LIN {X 0,Y 356.763,Z 514.388,A -85,B 0,C 180,E1 -13395.162,E2 -13395.162} C_VEL
LIN {X 0,Y 355.871,Z 522.553,A -85,B 0,C 180,E1 -13396.583,E2 -13396.583} C_VEL
LIN {X 0,Y 354.826,Z 530.602,A -85,B 0,C 180,E1 -13398.287,E2 -13398.287} C_VEL
LIN {X 0,Y 354.238,Z 536.073,A -85,B 0,C 180,E1 -13399.715,E2 -13399.715} C_VEL
LIN {X 0,Y 353.729,Z 541.453,A -85,B 0,C 180,E1 -13401.431,E2 -13401.431} C_VEL
LIN {X 0,Y 353.417,Z 545.66,A -85,B 0,C 180,E1 -13403.148,E2 -13403.148} C_VEL
LIN {X 0,Y 353.31,Z 547.883,A -85,B 0,C 180,E1 -13404.292,E2 -13404.292} C_VEL
LIN {X 0,Y 353.281,Z 549.633,A -85,B 0,C 180,E1 -13405.436,E2 -13405.436} C_VEL
LIN {X 0,Y 353.226,Z 550.976,A -85,B 0,C 180,E1 -13406.578,E2 -13406.578} C_VEL
LIN {X 0,Y 353.205,Z 551.922,A -85,B 0,C 180,E1 -13407.72,E2 -13407.72} C_VEL
LIN {X 0,Y 353.285,Z 552.443,A -85,B 0,C 180,E1 -13408.861,E2 -13408.861} C_VEL
LIN {X 0,Y 353.33,Z 552.542,A -85,B 0,C 180,E1 -13410,E2 -13410} C_VEL
LIN {X 0,Y 353.29,Z 552.246,A -85,B 0,C 180,E1 -13411.14,E2 -13411.14} C_VEL
LIN {X 0,Y 353.224,Z 551.556,A -85,B 0,C 180,E1 -13412.281,E2 -13412.281} C_VEL
LIN {X 0,Y 353.234,Z 550.435,A -85,B 0,C 180,E1 -13413.422,E2 -13413.422} C_VEL
LIN {X 0,Y 353.284,Z 548.872,A -85,B 0,C 180,E1 -13414.564,E2 -13414.564} C_VEL
LIN {X 0,Y 353.336,Z 545.71,A -85,B 0,C 180,E1 -13416.28,E2 -13416.28} C_VEL
LIN {X 0,Y 353.606,Z 541.468,A -85,B 0,C 180,E1 -13417.998,E2 -13417.998} C_VEL
LIN {X 0,Y 354.092,Z 535.01,A -85,B 0,C 180,E1 -13420.002,E2 -13420.002} C_VEL
LIN {X 0,Y 354.688,Z 527.935,A -85,B 0,C 180,E1 -13421.719,E2 -13421.719} C_VEL
LIN {X 0,Y 355.658,Z 519.093,A -85,B 0,C 180,E1 -13423.426,E2 -13423.426} C_VEL
LIN {X 0,Y 356.591,Z 510.04,A -85,B 0,C 180,E1 -13424.846,E2 -13424.846} C_VEL
LIN {X 0,Y 357.497,Z 500.082,A -85,B 0,C 180,E1 -13426.122,E2 -13426.122} C_VEL
LIN {X 0,Y 358.615,Z 489.083,A -85,B 0,C 180,E1 -13427.243,E2 -13427.243} C_VEL
LIN {X 0,Y 359.112,Z 482.478,A -85,B 0,C 180,E1 -13427.806,E2 -13427.806} C_VEL
LIN {X 0,Y 357.939,Z 470.567,A -85,B 0,C 180,E1 -13428.722,E2 -13428.722} C_VEL
LIN {X 0,Y 355.953,Z 457.17,A -85,B 0,C 180,E1 -13429.522,E2 -13429.522} C_VEL
LIN {X 0,Y 354.041,Z 446.07,A -85,B 0,C 180,E1 -13430.025,E2 -13430.025} C_VEL
LIN {X 0,Y 354.417,Z 439.879,A -85,B 0,C 180,E1 -13433.366,E2 -13433.366} C_VEL
LIN {X 0,Y 354.958,Z 433.091,A -85,B 0,C 180,E1 -13437.09,E2 -13437.09} C_VEL
LIN {X 0,Y 355.662,Z 426.292,A -85,B 0,C 180,E1 -13440.915,E2 -13440.915} C_VEL
LIN {X 0,Y 356.375,Z 419.492,A -85,B 0,C 180,E1 -13444.883,E2 -13444.883} C_VEL
LIN {X 0,Y 356.335,Z 416.053,A -85,B 0,C 180,E1 -13446.981,E2 -13446.981} C_VEL
LIN {X 0,Y 355.859,Z 411.923,A -85,B 0,C 180,E1 -13449.626,E2 -13449.626} C_VEL
LIN {X 0,Y 354.857,Z 406.322,A -85,B 0,C 180,E1 -13453.44,E2 -13453.44} C_VEL
LIN {X 0,Y 354.795,Z 406.29,A -85,B 0,C 180,E1 -13457.663,E2 -13457.663} C_VEL
LIN {X 0,Y 354.817,Z 406.286,A -85,B 0,C 180,E1 -13460.666,E2 -13460.666} C_VEL
LIN {X 0,Y 354.823,Z 406.284,A -85,B 0,C 180,E1 -13464.301,E2 -13464.301} C_VEL
LIN {X 0,Y 354.788,Z 406.29,A -85,B 0,C 180,E1 -13467.667,E2 -13467.667} C_VEL
LIN {X 0,Y 354.87,Z 406.28,A -85,B 0,C 180,E1 -13470.621,E2 -13470.621} C_VEL
LIN {X 0,Y 354.9,Z 406.274,A -85,B 0,C 180,E1 -13474.173,E2 -13474.173} C_VEL
LIN {X 0,Y 354.836,Z 406.283,A -85,B 0,C 180,E1 -13477.894,E2 -13477.894} C_VEL
LIN {X 0,Y 354.923,Z 406.272,A -85,B 0,C 180,E1 -13481.892,E2 -13481.892} C_VEL
LIN {X 0,Y 354.944,Z 406.269,A -85,B 0,C 180,E1 -13485.981,E2 -13485.981} C_VEL
LIN {X 0,Y 354.979,Z 406.265,A -85,B 0,C 180,E1 -13489.736,E2 -13489.736} C_VEL
LIN {X 0,Y 355.115,Z 406.248,A -85,B 0,C 180,E1 -13492.037,E2 -13492.037} C_VEL
LIN {X 0,Y 355.093,Z 406.251,A -85,B 0,C 180,E1 -13494.321,E2 -13494.321} C_VEL
LIN {X 0,Y 355.244,Z 406.232,A -85,B 0,C 180,E1 -13497.732,E2 -13497.732} C_VEL
LIN {X 0,Y 355.375,Z 406.215,A -85,B 0,C 180,E1 -13500,E2 -13500} C_VEL
LIN {X 0,Y 355.244,Z 406.232,A -85,B 0,C 180,E1 -13502.268,E2 -13502.268} C_VEL
LIN {X 0,Y 355.139,Z 406.25,A -85,B 0,C 180,E1 -13506.819,E2 -13506.819} C_VEL
LIN {X 0,Y 355.016,Z 406.264,A -85,B 0,C 180,E1 -13509.112,E2 -13509.112} C_VEL
LIN {X 0,Y 354.922,Z 406.275,A -85,B 0,C 180,E1 -13512.581,E2 -13512.581} C_VEL
LIN {X 0,Y 354.89,Z 406.276,A -85,B 0,C 180,E1 -13516.096,E2 -13516.096} C_VEL
LIN {X 0,Y 354.907,Z 406.277,A -85,B 0,C 180,E1 -13518.472,E2 -13518.472} C_VEL
LIN {X 0,Y 354.835,Z 406.283,A -85,B 0,C 180,E1 -13522.106,E2 -13522.106} C_VEL
LIN {X 0,Y 354.9,Z 406.274,A -85,B 0,C 180,E1 -13525.827,E2 -13525.827} C_VEL
LIN {X 0,Y 354.855,Z 406.28,A -85,B 0,C 180,E1 -13529.678,E2 -13529.678} C_VEL
LIN {X 0,Y 354.807,Z 406.286,A -85,B 0,C 180,E1 -13533.702,E2 -13533.702} C_VEL
LIN {X 0,Y 354.799,Z 406.291,A -85,B 0,C 180,E1 -13536.459,E2 -13536.459} C_VEL
LIN {X 0,Y 354.825,Z 406.284,A -85,B 0,C 180,E1 -13539.424,E2 -13539.424} C_VEL
LIN {X 0,Y 354.789,Z 406.292,A -85,B 0,C 180,E1 -13542.867,E2 -13542.867} C_VEL
LIN {X 0,Y 354.768,Z 406.293,A -85,B 0,C 180,E1 -13546.104,E2 -13546.104} C_VEL
LIN {X 0,Y 354.789,Z 406.289,A -85,B 0,C 180,E1 -13549.179,E2 -13549.179} C_VEL
LIN {X 0,Y 354.813,Z 406.29,A -85,B 0,C 180,E1 -13552.401,E2 -13552.401} C_VEL
LIN {X 0,Y 354.813,Z 406.287,A -85,B 0,C 180,E1 -13554.941,E2 -13554.941} C_VEL
LIN {X 0,Y 354.795,Z 406.292,A -85,B 0,C 180,E1 -13558.405,E2 -13558.405} C_VEL
LIN {X 0,Y 354.848,Z 406.281,A -85,B 0,C 180,E1 -13561.619,E2 -13561.619} C_VEL
LIN {X 0,Y 354.901,Z 406.278,A -85,B 0,C 180,E1 -13564.172,E2 -13564.172} C_VEL
LIN {X 0,Y 354.837,Z 406.283,A -85,B 0,C 180,E1 -13567.894,E2 -13567.894} C_VEL
LIN {X 0,Y 354.924,Z 406.273,A -85,B 0,C 180,E1 -13571.891,E2 -13571.891} C_VEL
LIN {X 0,Y 354.945,Z 406.271,A -85,B 0,C 180,E1 -13575.981,E2 -13575.981} C_VEL
LIN {X 0,Y 354.98,Z 406.265,A -85,B 0,C 180,E1 -13579.736,E2 -13579.736} C_VEL
LIN {X 0,Y 355.13,Z 406.249,A -85,B 0,C 180,E1 -13582.037,E2 -13582.037} C_VEL
LIN {X 0,Y 355.094,Z 406.255,A -85,B 0,C 180,E1 -13584.32,E2 -13584.32} C_VEL
LIN {X 0,Y 355.245,Z 406.233,A -85,B 0,C 180,E1 -13587.732,E2 -13587.732} C_VEL
LIN {X 0,Y 355.398,Z 406.216,A -85,B 0,C 180,E1 -13590,E2 -13590} C_VEL
LIN {X 0,Y 355.247,Z 406.237,A -85,B 0,C 180,E1 -13592.267,E2 -13592.267} C_VEL
LIN {X 0,Y 355.012,Z 406.261,A -85,B 0,C 180,E1 -13596.821,E2 -13596.821} C_VEL
LIN {X 0,Y 354.598,Z 406.315,A -85,B 0,C 180,E1 -13599.123,E2 -13599.123} C_VEL
LIN {X 0,Y 354.401,Z 408.438,A -85,B 0,C 180,E1 -13601.437,E2 -13601.437} C_VEL
LIN {X 0,Y 354.324,Z 410.917,A -85,B 0,C 180,E1 -13603.769,E2 -13603.769} C_VEL
LIN {X 0,Y 353.999,Z 415.198,A -85,B 0,C 180,E1 -13607.645,E2 -13607.645} C_VEL
LIN {X 0,Y 353.774,Z 418.936,A -85,B 0,C 180,E1 -13610.982,E2 -13610.982} C_VEL
LIN {X 0,Y 353.738,Z 421.29,A -85,B 0,C 180,E1 -13613.064,E2 -13613.064} C_VEL
LIN {X 0,Y 357.033,Z 435.378,A -85,B 0,C 180,E1 -13613.82,E2 -13613.82} C_VEL
LIN {X 0,Y 359.655,Z 448.278,A -85,B 0,C 180,E1 -13614.725,E2 -13614.725} C_VEL
LIN {X 0,Y 359.97,Z 452.375,A -85,B 0,C 180,E1 -13615.045,E2 -13615.045} C_VEL
LIN {X 0,Y 359.041,Z 463.653,A -85,B 0,C 180,E1 -13615.987,E2 -13615.987} C_VEL
LIN {X 0,Y 358.117,Z 474.495,A -85,B 0,C 180,E1 -13617.143,E2 -13617.143} C_VEL
LIN {X 0,Y 357.036,Z 484.857,A -85,B 0,C 180,E1 -13618.511,E2 -13618.511} C_VEL
LIN {X 0,Y 356.174,Z 493.935,A -85,B 0,C 180,E1 -13619.996,E2 -13619.996} C_VEL
LIN {X 0,Y 355.216,Z 502.345,A -85,B 0,C 180,E1 -13621.705,E2 -13621.705} C_VEL
LIN {X 0,Y 354.472,Z 509.826,A -85,B 0,C 180,E1 -13623.621,E2 -13623.621} C_VEL
LIN {X 0,Y 353.925,Z 515.495,A -85,B 0,C 180,E1 -13625.496,E2 -13625.496} C_VEL
LIN {X 0,Y 353.554,Z 519.696,A -85,B 0,C 180,E1 -13627.333,E2 -13627.333} C_VEL
LIN {X 0,Y 353.22,Z 523.205,A -85,B 0,C 180,E1 -13629.545,E2 -13629.545} C_VEL
LIN {X 0,Y 353.079,Z 524.676,A -85,B 0,C 180,E1 -13631.06,E2 -13631.06} C_VEL
LIN {X 0,Y 353.061,Z 525.477,A -85,B 0,C 180,E1 -13633.092,E2 -13633.092} C_VEL
LIN {X 0,Y 352.387,Z 525.561,A -85,B 0,C 180,E1 -13634.046,E2 -13634.046} C_VEL
LIN {X 0,Y 349.592,Z 525.045,A -85,B 0,C 180,E1 -13635.601,E2 -13635.601} C_VEL
LIN {X 0,Y 347.312,Z 524.205,A -85,B 0,C 180,E1 -13636.849,E2 -13636.849} C_VEL
LIN {X 0,Y 346.432,Z 523.164,A -85,B 0,C 180,E1 -13637.803,E2 -13637.803} C_VEL
LIN {X 0,Y 346.413,Z 522.725,A -85,B 0,C 180,E1 -13638.122,E2 -13638.122} C_VEL
LIN {X 0,Y 346.949,Z 518.902,A -85,B 0,C 180,E1 -13640.33,E2 -13640.33} C_VEL
LIN {X 0,Y 347.441,Z 514.693,A -85,B 0,C 180,E1 -13642.081,E2 -13642.081} C_VEL
LIN {X 0,Y 348.213,Z 509.279,A -85,B 0,C 180,E1 -13643.834,E2 -13643.834} C_VEL
LIN {X 0,Y 349.253,Z 501.981,A -85,B 0,C 180,E1 -13645.706,E2 -13645.706} C_VEL
LIN {X 0,Y 350.358,Z 493.618,A -85,B 0,C 180,E1 -13647.403,E2 -13647.403} C_VEL
LIN {X 0,Y 351.688,Z 483.939,A -85,B 0,C 180,E1 -13648.982,E2 -13648.982} C_VEL
LIN {X 0,Y 353.009,Z 473.091,A -85,B 0,C 180,E1 -13650.393,E2 -13650.393} C_VEL
LIN {X 0,Y 354.223,Z 461.722,A -85,B 0,C 180,E1 -13651.564,E2 -13651.564} C_VEL
LIN {X 0,Y 354.923,Z 454.745,A -85,B 0,C 180,E1 -13652.156,E2 -13652.156} C_VEL
LIN {X 0,Y 353.362,Z 445.433,A -85,B 0,C 180,E1 -13652.972,E2 -13652.972} C_VEL
LIN {X 0,Y 350.233,Z 433.278,A -85,B 0,C 180,E1 -13653.923,E2 -13653.923} C_VEL
LIN {X 0,Y 347.022,Z 422.964,A -85,B 0,C 180,E1 -13654.63,E2 -13654.63} C_VEL
LIN {X 0,Y 347.299,Z 418.94,A -85,B 0,C 180,E1 -13658.639,E2 -13658.639} C_VEL
LIN {X 0,Y 347.622,Z 415.352,A -85,B 0,C 180,E1 -13662.346,E2 -13662.346} C_VEL
LIN {X 0,Y 347.97,Z 411.993,A -85,B 0,C 180,E1 -13665.974,E2 -13665.974} C_VEL
LIN {X 0,Y 348.063,Z 408.92,A -85,B 0,C 180,E1 -13669.53,E2 -13669.53} C_VEL
LIN {X 0,Y 348.075,Z 407.133,A -85,B 0,C 180,E1 -13671.875,E2 -13671.875} C_VEL
LIN {X 0,Y 348.064,Z 407.131,A -85,B 0,C 180,E1 -13674.206,E2 -13674.206} C_VEL
LIN {X 0,Y 348.205,Z 407.115,A -85,B 0,C 180,E1 -13677.687,E2 -13677.687} C_VEL
LIN {X 0,Y 348.365,Z 407.093,A -85,B 0,C 180,E1 -13680,E2 -13680} C_VEL
LIN {X 0,Y 348.204,Z 407.11,A -85,B 0,C 180,E1 -13682.314,E2 -13682.314} C_VEL
LIN {X 0,Y 348.102,Z 407.126,A -85,B 0,C 180,E1 -13686.958,E2 -13686.958} C_VEL
LIN {X 0,Y 347.963,Z 407.142,A -85,B 0,C 180,E1 -13689.299,E2 -13689.299} C_VEL
LIN {X 0,Y 347.886,Z 407.153,A -85,B 0,C 180,E1 -13692.84,E2 -13692.84} C_VEL
LIN {X 0,Y 347.835,Z 407.16,A -85,B 0,C 180,E1 -13696.432,E2 -13696.432} C_VEL
LIN {X 0,Y 347.852,Z 407.156,A -85,B 0,C 180,E1 -13698.861,E2 -13698.861} C_VEL
LIN {X 0,Y 347.771,Z 407.167,A -85,B 0,C 180,E1 -13702.58,E2 -13702.58} C_VEL
LIN {X 0,Y 347.809,Z 407.162,A -85,B 0,C 180,E1 -13705.109,E2 -13705.109} C_VEL
LIN {X 0,Y 347.809,Z 407.163,A -85,B 0,C 180,E1 -13707.694,E2 -13707.694} C_VEL
LIN {X 0,Y 347.761,Z 407.168,A -85,B 0,C 180,E1 -13710.347,E2 -13710.347} C_VEL
LIN {X 0,Y 347.742,Z 407.171,A -85,B 0,C 180,E1 -13714.464,E2 -13714.464} C_VEL
LIN {X 0,Y 347.777,Z 407.169,A -85,B 0,C 180,E1 -13717.99,E2 -13717.99} C_VEL
LIN {X 0,Y 347.764,Z 407.171,A -85,B 0,C 180,E1 -13721.828,E2 -13721.828} C_VEL
LIN {X 0,Y 347.778,Z 407.283,A -85,B 0,C 180,E1 -13722.963,E2 -13722.963} C_VEL
LIN {X 0,Y 348.497,Z 411.314,A -85,B 0,C 180,E1 -13726.713,E2 -13726.713} C_VEL
LIN {X 0,Y 349.142,Z 415.165,A -85,B 0,C 180,E1 -13729.9,E2 -13729.9} C_VEL
LIN {X 0,Y 349.675,Z 419.167,A -85,B 0,C 180,E1 -13732.919,E2 -13732.919} C_VEL
LIN {X 0,Y 349.503,Z 423.291,A -85,B 0,C 180,E1 -13735.735,E2 -13735.735} C_VEL
LIN {X 0,Y 348.599,Z 429.618,A -85,B 0,C 180,E1 -13739.735,E2 -13739.735} C_VEL
LIN {X 0,Y 347.89,Z 436.102,A -85,B 0,C 180,E1 -13743.613,E2 -13743.613} C_VEL
LIN {X 0,Y 347.341,Z 442.681,A -85,B 0,C 180,E1 -13747.392,E2 -13747.392} C_VEL
LIN {X 0,Y 347.201,Z 444.613,A -85,B 0,C 180,E1 -13748.408,E2 -13748.408} C_VEL
LIN {X 0,Y 350.304,Z 458.15,A -85,B 0,C 180,E1 -13749.191,E2 -13749.191} C_VEL
LIN {X 0,Y 352.434,Z 470.851,A -85,B 0,C 180,E1 -13750.101,E2 -13750.101} C_VEL
LIN {X 0,Y 353.332,Z 482.24,A -85,B 0,C 180,E1 -13751.055,E2 -13751.055} C_VEL
LIN {X 0,Y 353.175,Z 487.99,A -85,B 0,C 180,E1 -13751.585,E2 -13751.585} C_VEL
LIN {X 0,Y 351.873,Z 498.895,A -85,B 0,C 180,E1 -13752.717,E2 -13752.717} C_VEL
LIN {X 0,Y 350.628,Z 508.537,A -85,B 0,C 180,E1 -13753.962,E2 -13753.962} C_VEL
LIN {X 0,Y 349.561,Z 517.851,A -85,B 0,C 180,E1 -13755.445,E2 -13755.445} C_VEL
LIN {X 0,Y 348.374,Z 526.733,A -85,B 0,C 180,E1 -13757.179,E2 -13757.179} C_VEL
LIN {X 0,Y 347.438,Z 533.896,A -85,B 0,C 180,E1 -13758.921,E2 -13758.921} C_VEL
LIN {X 0,Y 346.854,Z 539.65,A -85,B 0,C 180,E1 -13760.672,E2 -13760.672} C_VEL
LIN {X 0,Y 346.464,Z 544.204,A -85,B 0,C 180,E1 -13762.424,E2 -13762.424} C_VEL
LIN {X 0,Y 346.23,Z 547.676,A -85,B 0,C 180,E1 -13764.175,E2 -13764.175} C_VEL
LIN {X 0,Y 346.179,Z 549.414,A -85,B 0,C 180,E1 -13765.343,E2 -13765.343} C_VEL
LIN {X 0,Y 346.15,Z 550.746,A -85,B 0,C 180,E1 -13766.508,E2 -13766.508} C_VEL
LIN {X 0,Y 346.114,Z 551.679,A -85,B 0,C 180,E1 -13767.673,E2 -13767.673} C_VEL
LIN {X 0,Y 346.186,Z 552.174,A -85,B 0,C 180,E1 -13768.837,E2 -13768.837} C_VEL
LIN {X 0,Y 346.235,Z 552.261,A -85,B 0,C 180,E1 -13770,E2 -13770} C_VEL
LIN {X 0,Y 346.192,Z 551.951,A -85,B 0,C 180,E1 -13771.164,E2 -13771.164} C_VEL
LIN {X 0,Y 346.132,Z 551.247,A -85,B 0,C 180,E1 -13772.328,E2 -13772.328} C_VEL
LIN {X 0,Y 346.157,Z 550.098,A -85,B 0,C 180,E1 -13773.492,E2 -13773.492} C_VEL
LIN {X 0,Y 346.174,Z 547.182,A -85,B 0,C 180,E1 -13775.463,E2 -13775.463} C_VEL
LIN {X 0,Y 346.444,Z 542.612,A -85,B 0,C 180,E1 -13777.577,E2 -13777.577} C_VEL
LIN {X 0,Y 346.788,Z 537.556,A -85,B 0,C 180,E1 -13779.331,E2 -13779.331} C_VEL
LIN {X 0,Y 347.323,Z 531.186,A -85,B 0,C 180,E1 -13781.083,E2 -13781.083} C_VEL
LIN {X 0,Y 348.226,Z 523.209,A -85,B 0,C 180,E1 -13782.827,E2 -13782.827} C_VEL
LIN {X 0,Y 349.088,Z 515.082,A -85,B 0,C 180,E1 -13784.278,E2 -13784.278} C_VEL
LIN {X 0,Y 350.014,Z 505.606,A -85,B 0,C 180,E1 -13785.668,E2 -13785.668} C_VEL
LIN {X 0,Y 351.055,Z 495.486,A -85,B 0,C 180,E1 -13786.875,E2 -13786.875} C_VEL
LIN {X 0,Y 352.084,Z 485.062,A -85,B 0,C 180,E1 -13787.873,E2 -13787.873} C_VEL
LIN {X 0,Y 351.589,Z 476.667,A -85,B 0,C 180,E1 -13788.577,E2 -13788.577} C_VEL
LIN {X 0,Y 350.033,Z 464.231,A -85,B 0,C 180,E1 -13789.458,E2 -13789.458} C_VEL
LIN {X 0,Y 347.82,Z 450.648,A -85,B 0,C 180,E1 -13790.182,E2 -13790.182} C_VEL
LIN {X 0,Y 347.013,Z 445.844,A -85,B 0,C 180,E1 -13790.391,E2 -13790.391} C_VEL
LIN {X 0,Y 347.494,Z 438.444,A -85,B 0,C 180,E1 -13794.478,E2 -13794.478} C_VEL
LIN {X 0,Y 348.096,Z 431.644,A -85,B 0,C 180,E1 -13798.325,E2 -13798.325} C_VEL
LIN {X 0,Y 348.685,Z 425.984,A -85,B 0,C 180,E1 -13801.604,E2 -13801.604} C_VEL
LIN {X 0,Y 349.34,Z 420.319,A -85,B 0,C 180,E1 -13804.986,E2 -13804.986} C_VEL
LIN {X 0,Y 349.31,Z 416.89,A -85,B 0,C 180,E1 -13807.128,E2 -13807.128} C_VEL
LIN {X 0,Y 348.738,Z 412.487,A -85,B 0,C 180,E1 -13810.021,E2 -13810.021} C_VEL
LIN {X 0,Y 347.84,Z 407.486,A -85,B 0,C 180,E1 -13813.5,E2 -13813.5} C_VEL
LIN {X 0,Y 347.759,Z 407.169,A -85,B 0,C 180,E1 -13813.771,E2 -13813.771} C_VEL
LIN {X 0,Y 347.727,Z 407.171,A -85,B 0,C 180,E1 -13816.686,E2 -13816.686} C_VEL
LIN {X 0,Y 347.748,Z 407.165,A -85,B 0,C 180,E1 -13820.173,E2 -13820.173} C_VEL
LIN {X 0,Y 347.763,Z 407.165,A -85,B 0,C 180,E1 -13822.679,E2 -13822.679} C_VEL
LIN {X 0,Y 347.75,Z 407.165,A -85,B 0,C 180,E1 -13825.956,E2 -13825.956} C_VEL
LIN {X 0,Y 347.765,Z 407.165,A -85,B 0,C 180,E1 -13829.653,E2 -13829.653} C_VEL
LIN {X 0,Y 347.852,Z 407.155,A -85,B 0,C 180,E1 -13832.745,E2 -13832.745} C_VEL
LIN {X 0,Y 347.79,Z 407.16,A -85,B 0,C 180,E1 -13836.162,E2 -13836.162} C_VEL
LIN {X 0,Y 347.814,Z 407.157,A -85,B 0,C 180,E1 -13839.909,E2 -13839.909} C_VEL
LIN {X 0,Y 347.867,Z 407.151,A -85,B 0,C 180,E1 -13842.359,E2 -13842.359} C_VEL
LIN {X 0,Y 347.898,Z 407.146,A -85,B 0,C 180,E1 -13845.971,E2 -13845.971} C_VEL
LIN {X 0,Y 347.929,Z 407.144,A -85,B 0,C 180,E1 -13849.526,E2 -13849.526} C_VEL
LIN {X 0,Y 348.075,Z 407.125,A -85,B 0,C 180,E1 -13851.875,E2 -13851.875} C_VEL
LIN {X 0,Y 348.068,Z 407.126,A -85,B 0,C 180,E1 -13854.206,E2 -13854.206} C_VEL
LIN {X 0,Y 348.206,Z 407.109,A -85,B 0,C 180,E1 -13857.686,E2 -13857.686} C_VEL
LIN {X 0,Y 348.326,Z 407.093,A -85,B 0,C 180,E1 -13860,E2 -13860} C_VEL
LIN {X 0,Y 348.206,Z 407.109,A -85,B 0,C 180,E1 -13862.313,E2 -13862.313} C_VEL
LIN {X 0,Y 348.107,Z 407.126,A -85,B 0,C 180,E1 -13866.958,E2 -13866.958} C_VEL
LIN {X 0,Y 347.968,Z 407.14,A -85,B 0,C 180,E1 -13869.298,E2 -13869.298} C_VEL
LIN {X 0,Y 347.89,Z 407.153,A -85,B 0,C 180,E1 -13872.839,E2 -13872.839} C_VEL
LIN {X 0,Y 347.84,Z 407.156,A -85,B 0,C 180,E1 -13876.431,E2 -13876.431} C_VEL
LIN {X 0,Y 347.857,Z 407.157,A -85,B 0,C 180,E1 -13878.86,E2 -13878.86} C_VEL
LIN {X 0,Y 347.775,Z 407.166,A -85,B 0,C 180,E1 -13882.579,E2 -13882.579} C_VEL
LIN {X 0,Y 347.813,Z 407.16,A -85,B 0,C 180,E1 -13885.108,E2 -13885.108} C_VEL
LIN {X 0,Y 347.812,Z 407.157,A -85,B 0,C 180,E1 -13887.694,E2 -13887.694} C_VEL
LIN {X 0,Y 347.765,Z 407.166,A -85,B 0,C 180,E1 -13890.346,E2 -13890.346} C_VEL
LIN {X 0,Y 347.745,Z 407.169,A -85,B 0,C 180,E1 -13894.464,E2 -13894.464} C_VEL
LIN {X 0,Y 347.774,Z 407.162,A -85,B 0,C 180,E1 -13897.989,E2 -13897.989} C_VEL
LIN {X 0,Y 347.751,Z 407.165,A -85,B 0,C 180,E1 -13901.83,E2 -13901.83} C_VEL
LIN {X 0,Y 347.706,Z 407.173,A -85,B 0,C 180,E1 -13905.027,E2 -13905.027} C_VEL
LIN {X 0,Y 347.751,Z 407.169,A -85,B 0,C 180,E1 -13908.397,E2 -13908.397} C_VEL
LIN {X 0,Y 347.778,Z 407.163,A -85,B 0,C 180,E1 -13912.011,E2 -13912.011} C_VEL
LIN {X 0,Y 347.746,Z 407.165,A -85,B 0,C 180,E1 -13915.536,E2 -13915.536} C_VEL
LIN {X 0,Y 347.746,Z 407.169,A -85,B 0,C 180,E1 -13918.3,E2 -13918.3} C_VEL
LIN {X 0,Y 347.78,Z 407.163,A -85,B 0,C 180,E1 -13920.988,E2 -13920.988} C_VEL
LIN {X 0,Y 347.832,Z 407.155,A -85,B 0,C 180,E1 -13923.608,E2 -13923.608} C_VEL
LIN {X 0,Y 347.791,Z 407.163,A -85,B 0,C 180,E1 -13926.162,E2 -13926.162} C_VEL
LIN {X 0,Y 347.815,Z 407.158,A -85,B 0,C 180,E1 -13929.909,E2 -13929.909} C_VEL
LIN {X 0,Y 347.868,Z 407.156,A -85,B 0,C 180,E1 -13932.359,E2 -13932.359} C_VEL
LIN {X 0,Y 347.899,Z 407.149,A -85,B 0,C 180,E1 -13935.971,E2 -13935.971} C_VEL
LIN {X 0,Y 347.93,Z 407.142,A -85,B 0,C 180,E1 -13939.525,E2 -13939.525} C_VEL
LIN {X 0,Y 348.11,Z 407.121,A -85,B 0,C 180,E1 -13943.042,E2 -13943.042} C_VEL
LIN {X 0,Y 348.207,Z 407.109,A -85,B 0,C 180,E1 -13947.686,E2 -13947.686} C_VEL
LIN {X 0,Y 348.346,Z 407.094,A -85,B 0,C 180,E1 -13950,E2 -13950} C_VEL
LIN {X 0,Y 348.209,Z 407.113,A -85,B 0,C 180,E1 -13952.313,E2 -13952.313} C_VEL
LIN {X 0,Y 348.02,Z 407.133,A -85,B 0,C 180,E1 -13955.795,E2 -13955.795} C_VEL
LIN {X 0,Y 347.736,Z 407.172,A -85,B 0,C 180,E1 -13958.133,E2 -13958.133} C_VEL
LIN {X 0,Y 347.524,Z 407.196,A -85,B 0,C 180,E1 -13959.31,E2 -13959.31} C_VEL
LIN {X 0,Y 347.326,Z 410.762,A -85,B 0,C 180,E1 -13962.86,E2 -13962.86} C_VEL
LIN {X 0,Y 346.985,Z 414.642,A -85,B 0,C 180,E1 -13966.472,E2 -13966.472} C_VEL
LIN {X 0,Y 346.739,Z 418.725,A -85,B 0,C 180,E1 -13970.155,E2 -13970.155} C_VEL
LIN {X 0,Y 346.638,Z 421.563,A -85,B 0,C 180,E1 -13972.696,E2 -13972.696} C_VEL
LIN {X 0,Y 350.042,Z 435.676,A -85,B 0,C 180,E1 -13973.478,E2 -13973.478} C_VEL
LIN {X 0,Y 352.692,Z 448.785,A -85,B 0,C 180,E1 -13974.423,E2 -13974.423} C_VEL
LIN {X 0,Y 353.121,Z 453.224,A -85,B 0,C 180,E1 -13974.783,E2 -13974.783} C_VEL
LIN {X 0,Y 352.177,Z 464.157,A -85,B 0,C 180,E1 -13975.724,E2 -13975.724} C_VEL
LIN {X 0,Y 351.175,Z 475.125,A -85,B 0,C 180,E1 -13976.922,E2 -13976.922} C_VEL
LIN {X 0,Y 350.016,Z 485.905,A -85,B 0,C 180,E1 -13978.388,E2 -13978.388} C_VEL
LIN {X 0,Y 349.057,Z 495.466,A -85,B 0,C 180,E1 -13980.029,E2 -13980.029} C_VEL
LIN {X 0,Y 348.144,Z 503.166,A -85,B 0,C 180,E1 -13981.658,E2 -13981.658} C_VEL
LIN {X 0,Y 347.429,Z 510.191,A -85,B 0,C 180,E1 -13983.51,E2 -13983.51} C_VEL
LIN {X 0,Y 346.911,Z 515.218,A -85,B 0,C 180,E1 -13985.184,E2 -13985.184} C_VEL
LIN {X 0,Y 346.556,Z 518.912,A -85,B 0,C 180,E1 -13986.744,E2 -13986.744} C_VEL
LIN {X 0,Y 346.328,Z 521.77,A -85,B 0,C 180,E1 -13988.302,E2 -13988.302} C_VEL
LIN {X 0,Y 346.025,Z 524.54,A -85,B 0,C 180,E1 -13990.536,E2 -13990.536} C_VEL
LIN {X 0,Y 345.996,Z 525.535,A -85,B 0,C 180,E1 -13992.09,E2 -13992.09} C_VEL
LIN {X 0,Y 345.984,Z 525.845,A -85,B 0,C 180,E1 -13993.68,E2 -13993.68} C_VEL
LIN {X 0,Y 346.028,Z 525.406,A -85,B 0,C 180,E1 -13995.304,E2 -13995.304} C_VEL
LIN {X 0,Y 346.213,Z 524.128,A -85,B 0,C 180,E1 -13996.951,E2 -13996.951} C_VEL
LIN {X 0,Y 346.413,Z 522.725,A -85,B 0,C 180,E1 -13998.122,E2 -13998.122} C_VEL
LIN {X 0,Y 345.957,Z 521.356,A -85,B 0,C 180,E1 -13999.069,E2 -13999.069} C_VEL
LIN {X 0,Y 343.495,Z 518.707,A -85,B 0,C 180,E1 -14000.606,E2 -14000.606} C_VEL
LIN {X 0,Y 341.465,Z 516.174,A -85,B 0,C 180,E1 -14001.823,E2 -14001.823} C_VEL
LIN {X 0,Y 340.763,Z 513.872,A -85,B 0,C 180,E1 -14002.732,E2 -14002.732} C_VEL
LIN {X 0,Y 340.8,Z 512.997,A -85,B 0,C 180,E1 -14003.03,E2 -14003.03} C_VEL
LIN {X 0,Y 341.628,Z 507.032,A -85,B 0,C 180,E1 -14004.829,E2 -14004.829} C_VEL
LIN {X 0,Y 342.559,Z 500.753,A -85,B 0,C 180,E1 -14006.362,E2 -14006.362} C_VEL
LIN {X 0,Y 343.648,Z 493.227,A -85,B 0,C 180,E1 -14007.878,E2 -14007.878} C_VEL
LIN {X 0,Y 345.004,Z 484.056,A -85,B 0,C 180,E1 -14009.385,E2 -14009.385} C_VEL
LIN {X 0,Y 346.32,Z 473.681,A -85,B 0,C 180,E1 -14010.762,E2 -14010.762} C_VEL
LIN {X 0,Y 347.596,Z 462.356,A -85,B 0,C 180,E1 -14011.96,E2 -14011.96} C_VEL
LIN {X 0,Y 348.27,Z 456.14,A -85,B 0,C 180,E1 -14012.504,E2 -14012.504} C_VEL
LIN {X 0,Y 346.435,Z 445.399,A -85,B 0,C 180,E1 -14013.493,E2 -14013.493} C_VEL
LIN {X 0,Y 343.142,Z 433.06,A -85,B 0,C 180,E1 -14014.485,E2 -14014.485} C_VEL
LIN {X 0,Y 339.984,Z 423.278,A -85,B 0,C 180,E1 -14015.195,E2 -14015.195} C_VEL
LIN {X 0,Y 340.315,Z 419.114,A -85,B 0,C 180,E1 -14019.447,E2 -14019.447} C_VEL
LIN {X 0,Y 340.665,Z 415.59,A -85,B 0,C 180,E1 -14023.213,E2 -14023.213} C_VEL
LIN {X 0,Y 340.982,Z 412.316,A -85,B 0,C 180,E1 -14026.896,E2 -14026.896} C_VEL
LIN {X 0,Y 341.072,Z 409.317,A -85,B 0,C 180,E1 -14030.512,E2 -14030.512} C_VEL
LIN {X 0,Y 341.083,Z 408.364,A -85,B 0,C 180,E1 -14031.707,E2 -14031.707} C_VEL
LIN {X 0,Y 341.073,Z 408.002,A -85,B 0,C 180,E1 -14032.898,E2 -14032.898} C_VEL
LIN {X 0,Y 341.166,Z 407.991,A -85,B 0,C 180,E1 -14037.639,E2 -14037.639} C_VEL
LIN {X 0,Y 341.314,Z 407.972,A -85,B 0,C 180,E1 -14040,E2 -14040} C_VEL
LIN {X 0,Y 341.166,Z 407.987,A -85,B 0,C 180,E1 -14042.361,E2 -14042.361} C_VEL
LIN {X 0,Y 341.072,Z 408.001,A -85,B 0,C 180,E1 -14047.102,E2 -14047.102} C_VEL
LIN {X 0,Y 340.867,Z 408.026,A -85,B 0,C 180,E1 -14050.694,E2 -14050.694} C_VEL
LIN {X 0,Y 340.859,Z 408.028,A -85,B 0,C 180,E1 -14054.325,E2 -14054.325} C_VEL
LIN {X 0,Y 340.834,Z 408.03,A -85,B 0,C 180,E1 -14058.467,E2 -14058.467} C_VEL
LIN {X 0,Y 340.75,Z 408.041,A -85,B 0,C 180,E1 -14061.857,E2 -14061.857} C_VEL
LIN {X 0,Y 340.77,Z 408.039,A -85,B 0,C 180,E1 -14065.665,E2 -14065.665} C_VEL
LIN {X 0,Y 340.739,Z 408.042,A -85,B 0,C 180,E1 -14068.32,E2 -14068.32} C_VEL
LIN {X 0,Y 340.701,Z 408.048,A -85,B 0,C 180,E1 -14071.045,E2 -14071.045} C_VEL
LIN {X 0,Y 340.716,Z 408.048,A -85,B 0,C 180,E1 -14075.279,E2 -14075.279} C_VEL
LIN {X 0,Y 340.717,Z 408.049,A -85,B 0,C 180,E1 -14078.389,E2 -14078.389} C_VEL
LIN {X 0,Y 340.715,Z 408.051,A -85,B 0,C 180,E1 -14082.189,E2 -14082.189} C_VEL
LIN {X 0,Y 341.42,Z 412.084,A -85,B 0,C 180,E1 -14086.093,E2 -14086.093} C_VEL
LIN {X 0,Y 342.063,Z 416.006,A -85,B 0,C 180,E1 -14089.482,E2 -14089.482} C_VEL
LIN {X 0,Y 342.554,Z 419.218,A -85,B 0,C 180,E1 -14092.013,E2 -14092.013} C_VEL
LIN {X 0,Y 342.665,Z 422.257,A -85,B 0,C 180,E1 -14094.231,E2 -14094.231} C_VEL
LIN {X 0,Y 342.018,Z 427.441,A -85,B 0,C 180,E1 -14097.707,E2 -14097.707} C_VEL
LIN {X 0,Y 341.166,Z 433.826,A -85,B 0,C 180,E1 -14101.72,E2 -14101.72} C_VEL
LIN {X 0,Y 340.517,Z 440.346,A -85,B 0,C 180,E1 -14105.621,E2 -14105.621} C_VEL
LIN {X 0,Y 340.245,Z 444.312,A -85,B 0,C 180,E1 -14107.857,E2 -14107.857} C_VEL
LIN {X 0,Y 343.432,Z 457.952,A -85,B 0,C 180,E1 -14108.677,E2 -14108.677} C_VEL
LIN {X 0,Y 345.501,Z 470.026,A -85,B 0,C 180,E1 -14109.572,E2 -14109.572} C_VEL
LIN {X 0,Y 346.495,Z 481.283,A -85,B 0,C 180,E1 -14110.543,E2 -14110.543} C_VEL
LIN {X 0,Y 346.453,Z 488.312,A -85,B 0,C 180,E1 -14111.215,E2 -14111.215} C_VEL
LIN {X 0,Y 345.101,Z 499.072,A -85,B 0,C 180,E1 -14112.367,E2 -14112.367} C_VEL
LIN {X 0,Y 343.778,Z 508.808,A -85,B 0,C 180,E1 -14113.661,E2 -14113.661} C_VEL
LIN {X 0,Y 342.669,Z 517.882,A -85,B 0,C 180,E1 -14115.146,E2 -14115.146} C_VEL
LIN {X 0,Y 341.439,Z 526.715,A -85,B 0,C 180,E1 -14116.914,E2 -14116.914} C_VEL
LIN {X 0,Y 340.43,Z 533.811,A -85,B 0,C 180,E1 -14118.69,E2 -14118.69} C_VEL
LIN {X 0,Y 339.808,Z 539.516,A -85,B 0,C 180,E1 -14120.477,E2 -14120.477} C_VEL
LIN {X 0,Y 339.395,Z 544.03,A -85,B 0,C 180,E1 -14122.265,E2 -14122.265} C_VEL
LIN {X 0,Y 339.135,Z 547.558,A -85,B 0,C 180,E1 -14124.11,E2 -14124.11} C_VEL
LIN {X 0,Y 339.074,Z 550.517,A -85,B 0,C 180,E1 -14126.435,E2 -14126.435} C_VEL
LIN {X 0,Y 339.027,Z 551.432,A -85,B 0,C 180,E1 -14127.624,E2 -14127.624} C_VEL
LIN {X 0,Y 339.087,Z 551.905,A -85,B 0,C 180,E1 -14128.813,E2 -14128.813} C_VEL
LIN {X 0,Y 339.14,Z 551.979,A -85,B 0,C 180,E1 -14130,E2 -14130} C_VEL
LIN {X 0,Y 339.094,Z 551.657,A -85,B 0,C 180,E1 -14131.188,E2 -14131.188} C_VEL
LIN {X 0,Y 339.043,Z 550.935,A -85,B 0,C 180,E1 -14132.376,E2 -14132.376} C_VEL
LIN {X 0,Y 339.082,Z 549.762,A -85,B 0,C 180,E1 -14133.565,E2 -14133.565} C_VEL
LIN {X 0,Y 339.094,Z 548.167,A -85,B 0,C 180,E1 -14134.756,E2 -14134.756} C_VEL
LIN {X 0,Y 339.194,Z 544.942,A -85,B 0,C 180,E1 -14136.544,E2 -14136.544} C_VEL
LIN {X 0,Y 339.477,Z 540.631,A -85,B 0,C 180,E1 -14138.333,E2 -14138.333} C_VEL
LIN {X 0,Y 340.043,Z 534.092,A -85,B 0,C 180,E1 -14140.419,E2 -14140.419} C_VEL
LIN {X 0,Y 340.749,Z 526.893,A -85,B 0,C 180,E1 -14142.205,E2 -14142.205} C_VEL
LIN {X 0,Y 341.738,Z 517.943,A -85,B 0,C 180,E1 -14143.984,E2 -14143.984} C_VEL
LIN {X 0,Y 342.687,Z 508.763,A -85,B 0,C 180,E1 -14145.463,E2 -14145.463} C_VEL
LIN {X 0,Y 343.785,Z 498.595,A -85,B 0,C 180,E1 -14146.784,E2 -14146.784} C_VEL
LIN {X 0,Y 345,Z 487.387,A -85,B 0,C 180,E1 -14147.946,E2 -14147.946} C_VEL
LIN {X 0,Y 345.118,Z 482.363,A -85,B 0,C 180,E1 -14148.4,E2 -14148.4} C_VEL
LIN {X 0,Y 343.888,Z 470.053,A -85,B 0,C 180,E1 -14149.397,E2 -14149.397} C_VEL
LIN {X 0,Y 341.902,Z 456.815,A -85,B 0,C 180,E1 -14150.233,E2 -14150.233} C_VEL
LIN {X 0,Y 339.957,Z 445.557,A -85,B 0,C 180,E1 -14150.783,E2 -14150.783} C_VEL
LIN {X 0,Y 340.457,Z 438.598,A -85,B 0,C 180,E1 -14154.73,E2 -14154.73} C_VEL
LIN {X 0,Y 341.157,Z 431.305,A -85,B 0,C 180,E1 -14158.955,E2 -14158.955} C_VEL
LIN {X 0,Y 341.771,Z 425.657,A -85,B 0,C 180,E1 -14162.32,E2 -14162.32} C_VEL
LIN {X 0,Y 342.33,Z 421.121,A -85,B 0,C 180,E1 -14165.088,E2 -14165.088} C_VEL
LIN {X 0,Y 342.165,Z 416.546,A -85,B 0,C 180,E1 -14168.039,E2 -14168.039} C_VEL
LIN {X 0,Y 341.427,Z 411.918,A -85,B 0,C 180,E1 -14171.201,E2 -14171.201} C_VEL
LIN {X 0,Y 340.711,Z 408.047,A -85,B 0,C 180,E1 -14173.999,E2 -14173.999} C_VEL
LIN {X 0,Y 340.7,Z 408.043,A -85,B 0,C 180,E1 -14177.955,E2 -14177.955} C_VEL
LIN {X 0,Y 340.734,Z 408.04,A -85,B 0,C 180,E1 -14181.773,E2 -14181.773} C_VEL
LIN {X 0,Y 340.724,Z 408.042,A -85,B 0,C 180,E1 -14185.595,E2 -14185.595} C_VEL
LIN {X 0,Y 340.705,Z 408.046,A -85,B 0,C 180,E1 -14188.956,E2 -14188.956} C_VEL
LIN {X 0,Y 340.779,Z 408.034,A -85,B 0,C 180,E1 -14192.474,E2 -14192.474} C_VEL
LIN {X 0,Y 340.757,Z 408.037,A -85,B 0,C 180,E1 -14195.638,E2 -14195.638} C_VEL
LIN {X 0,Y 340.746,Z 408.04,A -85,B 0,C 180,E1 -14199.474,E2 -14199.474} C_VEL
LIN {X 0,Y 340.859,Z 408.023,A -85,B 0,C 180,E1 -14201.984,E2 -14201.984} C_VEL
LIN {X 0,Y 340.87,Z 408.022,A -85,B 0,C 180,E1 -14205.705,E2 -14205.705} C_VEL
LIN {X 0,Y 340.872,Z 408.025,A -85,B 0,C 180,E1 -14209.306,E2 -14209.306} C_VEL
LIN {X 0,Y 341.076,Z 408.001,A -85,B 0,C 180,E1 -14212.898,E2 -14212.898} C_VEL
LIN {X 0,Y 341.168,Z 407.985,A -85,B 0,C 180,E1 -14217.639,E2 -14217.639} C_VEL
LIN {X 0,Y 341.277,Z 407.971,A -85,B 0,C 180,E1 -14220,E2 -14220} C_VEL
LIN {X 0,Y 341.168,Z 407.986,A -85,B 0,C 180,E1 -14222.361,E2 -14222.361} C_VEL
LIN {X 0,Y 341.076,Z 408,A -85,B 0,C 180,E1 -14227.102,E2 -14227.102} C_VEL
LIN {X 0,Y 340.872,Z 408.026,A -85,B 0,C 180,E1 -14230.694,E2 -14230.694} C_VEL
LIN {X 0,Y 340.864,Z 408.024,A -85,B 0,C 180,E1 -14234.325,E2 -14234.325} C_VEL
LIN {X 0,Y 340.839,Z 408.028,A -85,B 0,C 180,E1 -14238.467,E2 -14238.467} C_VEL
LIN {X 0,Y 340.755,Z 408.036,A -85,B 0,C 180,E1 -14241.857,E2 -14241.857} C_VEL
LIN {X 0,Y 340.774,Z 408.034,A -85,B 0,C 180,E1 -14245.664,E2 -14245.664} C_VEL
LIN {X 0,Y 340.742,Z 408.04,A -85,B 0,C 180,E1 -14248.32,E2 -14248.32} C_VEL
LIN {X 0,Y 340.704,Z 408.045,A -85,B 0,C 180,E1 -14251.044,E2 -14251.044} C_VEL
LIN {X 0,Y 340.719,Z 408.042,A -85,B 0,C 180,E1 -14255.279,E2 -14255.279} C_VEL
LIN {X 0,Y 340.71,Z 408.045,A -85,B 0,C 180,E1 -14258.386,E2 -14258.386} C_VEL
LIN {X 0,Y 340.7,Z 408.044,A -85,B 0,C 180,E1 -14262.045,E2 -14262.045} C_VEL
LIN {X 0,Y 340.653,Z 408.051,A -85,B 0,C 180,E1 -14266.227,E2 -14266.227} C_VEL
LIN {X 0,Y 340.689,Z 408.044,A -85,B 0,C 180,E1 -14269.753,E2 -14269.753} C_VEL
LIN {X 0,Y 340.708,Z 408.043,A -85,B 0,C 180,E1 -14273.259,E2 -14273.259} C_VEL
LIN {X 0,Y 340.694,Z 408.046,A -85,B 0,C 180,E1 -14276.153,E2 -14276.153} C_VEL
LIN {X 0,Y 340.743,Z 408.042,A -85,B 0,C 180,E1 -14280.329,E2 -14280.329} C_VEL
LIN {X 0,Y 340.805,Z 408.031,A -85,B 0,C 180,E1 -14283.02,E2 -14283.02} C_VEL
LIN {X 0,Y 340.758,Z 408.036,A -85,B 0,C 180,E1 -14285.638,E2 -14285.638} C_VEL
LIN {X 0,Y 340.747,Z 408.037,A -85,B 0,C 180,E1 -14289.474,E2 -14289.474} C_VEL
LIN {X 0,Y 340.859,Z 408.025,A -85,B 0,C 180,E1 -14291.984,E2 -14291.984} C_VEL
LIN {X 0,Y 340.871,Z 408.022,A -85,B 0,C 180,E1 -14295.705,E2 -14295.705} C_VEL
LIN {X 0,Y 340.873,Z 408.021,A -85,B 0,C 180,E1 -14299.306,E2 -14299.306} C_VEL
LIN {X 0,Y 341.08,Z 407.997,A -85,B 0,C 180,E1 -14302.898,E2 -14302.898} C_VEL
LIN {X 0,Y 341.169,Z 407.985,A -85,B 0,C 180,E1 -14307.638,E2 -14307.638} C_VEL
LIN {X 0,Y 341.297,Z 407.972,A -85,B 0,C 180,E1 -14310,E2 -14310} C_VEL
LIN {X 0,Y 341.171,Z 407.99,A -85,B 0,C 180,E1 -14312.361,E2 -14312.361} C_VEL
LIN {X 0,Y 340.986,Z 408.01,A -85,B 0,C 180,E1 -14315.915,E2 -14315.915} C_VEL
LIN {X 0,Y 340.669,Z 408.052,A -85,B 0,C 180,E1 -14318.303,E2 -14318.303} C_VEL
LIN {X 0,Y 340.45,Z 408.143,A -85,B 0,C 180,E1 -14319.505,E2 -14319.505} C_VEL
LIN {X 0,Y 340.224,Z 412.619,A -85,B 0,C 180,E1 -14323.861,E2 -14323.861} C_VEL
LIN {X 0,Y 339.824,Z 417.111,A -85,B 0,C 180,E1 -14328.072,E2 -14328.072} C_VEL
LIN {X 0,Y 339.594,Z 421.791,A -85,B 0,C 180,E1 -14332.31,E2 -14332.31} C_VEL
LIN {X 0,Y 343.183,Z 436.842,A -85,B 0,C 180,E1 -14333.177,E2 -14333.177} C_VEL
LIN {X 0,Y 345.793,Z 449.684,A -85,B 0,C 180,E1 -14334.143,E2 -14334.143} C_VEL
LIN {X 0,Y 346.265,Z 454.013,A -85,B 0,C 180,E1 -14334.507,E2 -14334.507} C_VEL
LIN {X 0,Y 345.144,Z 466.139,A -85,B 0,C 180,E1 -14335.601,E2 -14335.601} C_VEL
LIN {X 0,Y 344.106,Z 477.122,A -85,B 0,C 180,E1 -14336.864,E2 -14336.864} C_VEL
LIN {X 0,Y 343.012,Z 486.765,A -85,B 0,C 180,E1 -14338.233,E2 -14338.233} C_VEL
LIN {X 0,Y 342.041,Z 496.158,A -85,B 0,C 180,E1 -14339.899,E2 -14339.899} C_VEL
LIN {X 0,Y 341.073,Z 504.062,A -85,B 0,C 180,E1 -14341.627,E2 -14341.627} C_VEL
LIN {X 0,Y 340.348,Z 510.989,A -85,B 0,C 180,E1 -14343.529,E2 -14343.529} C_VEL
LIN {X 0,Y 339.762,Z 516.284,A -85,B 0,C 180,E1 -14345.392,E2 -14345.392} C_VEL
LIN {X 0,Y 339.368,Z 520.755,A -85,B 0,C 180,E1 -14347.485,E2 -14347.485} C_VEL
LIN {X 0,Y 339.215,Z 522.308,A -85,B 0,C 180,E1 -14348.429,E2 -14348.429} C_VEL
LIN {X 0,Y 338.992,Z 524.282,A -85,B 0,C 180,E1 -14349.992,E2 -14349.992} C_VEL
LIN {X 0,Y 338.91,Z 525.632,A -85,B 0,C 180,E1 -14351.709,E2 -14351.709} C_VEL
LIN {X 0,Y 338.896,Z 526.14,A -85,B 0,C 180,E1 -14353.462,E2 -14353.462} C_VEL
LIN {X 0,Y 338.924,Z 525.779,A -85,B 0,C 180,E1 -14355.168,E2 -14355.168} C_VEL
LIN {X 0,Y 339.105,Z 524.625,A -85,B 0,C 180,E1 -14356.848,E2 -14356.848} C_VEL
LIN {X 0,Y 339.417,Z 522.706,A -85,B 0,C 180,E1 -14358.502,E2 -14358.502} C_VEL
LIN {X 0,Y 339.832,Z 520.03,A -85,B 0,C 180,E1 -14360.126,E2 -14360.126} C_VEL
LIN {X 0,Y 340.387,Z 515.576,A -85,B 0,C 180,E1 -14362.102,E2 -14362.102} C_VEL
LIN {X 0,Y 340.8,Z 512.997,A -85,B 0,C 180,E1 -14363.03,E2 -14363.03} C_VEL
LIN {X 0,Y 340.529,Z 510.357,A -85,B 0,C 180,E1 -14363.916,E2 -14363.916} C_VEL
LIN {X 0,Y 338.427,Z 505.772,A -85,B 0,C 180,E1 -14365.36,E2 -14365.36} C_VEL
LIN {X 0,Y 336.44,Z 500.622,A -85,B 0,C 180,E1 -14366.759,E2 -14366.759} C_VEL
LIN {X 0,Y 336.343,Z 497.036,A -85,B 0,C 180,E1 -14367.562,E2 -14367.562} C_VEL
LIN {X 0,Y 337.758,Z 488.113,A -85,B 0,C 180,E1 -14369.196,E2 -14369.196} C_VEL
LIN {X 0,Y 339.184,Z 478.213,A -85,B 0,C 180,E1 -14370.652,E2 -14370.652} C_VEL
LIN {X 0,Y 340.601,Z 466.804,A -85,B 0,C 180,E1 -14371.996,E2 -14371.996} C_VEL
LIN {X 0,Y 341.65,Z 456.873,A -85,B 0,C 180,E1 -14372.932,E2 -14372.932} C_VEL
LIN {X 0,Y 339.53,Z 445.45,A -85,B 0,C 180,E1 -14374.029,E2 -14374.029} C_VEL
LIN {X 0,Y 335.927,Z 432.479,A -85,B 0,C 180,E1 -14375.11,E2 -14375.11} C_VEL
LIN {X 0,Y 332.991,Z 423.608,A -85,B 0,C 180,E1 -14375.78,E2 -14375.78} C_VEL
LIN {X 0,Y 333.231,Z 420.532,A -85,B 0,C 180,E1 -14378.99,E2 -14378.99} C_VEL
LIN {X 0,Y 333.591,Z 416.973,A -85,B 0,C 180,E1 -14382.846,E2 -14382.846} C_VEL
LIN {X 0,Y 333.938,Z 413.681,A -85,B 0,C 180,E1 -14386.614,E2 -14386.614} C_VEL
LIN {X 0,Y 334.067,Z 410.678,A -85,B 0,C 180,E1 -14390.311,E2 -14390.311} C_VEL
LIN {X 0,Y 334.029,Z 408.88,A -85,B 0,C 180,E1 -14392.748,E2 -14392.748} C_VEL
LIN {X 0,Y 334.104,Z 408.871,A -85,B 0,C 180,E1 -14397.589,E2 -14397.589} C_VEL
LIN {X 0,Y 334.264,Z 408.85,A -85,B 0,C 180,E1 -14400,E2 -14400} C_VEL
LIN {X 0,Y 334.103,Z 408.866,A -85,B 0,C 180,E1 -14402.411,E2 -14402.411} C_VEL
LIN {X 0,Y 334.021,Z 408.88,A -85,B 0,C 180,E1 -14407.253,E2 -14407.253} C_VEL
LIN {X 0,Y 333.83,Z 408.903,A -85,B 0,C 180,E1 -14410.922,E2 -14410.922} C_VEL
LIN {X 0,Y 333.804,Z 408.906,A -85,B 0,C 180,E1 -14414.635,E2 -14414.635} C_VEL
LIN {X 0,Y 333.793,Z 408.907,A -85,B 0,C 180,E1 -14418.656,E2 -14418.656} C_VEL
LIN {X 0,Y 333.689,Z 408.92,A -85,B 0,C 180,E1 -14422.279,E2 -14422.279} C_VEL
LIN {X 0,Y 333.733,Z 408.915,A -85,B 0,C 180,E1 -14426.247,E2 -14426.247} C_VEL
LIN {X 0,Y 333.708,Z 408.919,A -85,B 0,C 180,E1 -14428.972,E2 -14428.972} C_VEL
LIN {X 0,Y 333.643,Z 408.927,A -85,B 0,C 180,E1 -14432.588,E2 -14432.588} C_VEL
LIN {X 0,Y 333.675,Z 408.925,A -85,B 0,C 180,E1 -14436.139,E2 -14436.139} C_VEL
LIN {X 0,Y 333.67,Z 408.927,A -85,B 0,C 180,E1 -14439.189,E2 -14439.189} C_VEL
LIN {X 0,Y 333.689,Z 409.013,A -85,B 0,C 180,E1 -14441.563,E2 -14441.563} C_VEL
LIN {X 0,Y 334.132,Z 411.693,A -85,B 0,C 180,E1 -14444.346,E2 -14444.346} C_VEL
LIN {X 0,Y 334.778,Z 415.395,A -85,B 0,C 180,E1 -14447.797,E2 -14447.797} C_VEL
LIN {X 0,Y 335.443,Z 419.265,A -85,B 0,C 180,E1 -14451.058,E2 -14451.058} C_VEL
LIN {X 0,Y 335.663,Z 421.421,A -85,B 0,C 180,E1 -14452.715,E2 -14452.715} C_VEL
LIN {X 0,Y 335.612,Z 424.189,A -85,B 0,C 180,E1 -14454.756,E2 -14454.756} C_VEL
LIN {X 0,Y 334.806,Z 429.51,A -85,B 0,C 180,E1 -14458.347,E2 -14458.347} C_VEL
LIN {X 0,Y 334.013,Z 435.901,A -85,B 0,C 180,E1 -14462.426,E2 -14462.426} C_VEL
LIN {X 0,Y 333.343,Z 442.408,A -85,B 0,C 180,E1 -14466.386,E2 -14466.386} C_VEL
LIN {X 0,Y 333.248,Z 443.834,A -85,B 0,C 180,E1 -14467.239,E2 -14467.239} C_VEL
LIN {X 0,Y 336.87,Z 459.175,A -85,B 0,C 180,E1 -14468.246,E2 -14468.246} C_VEL
LIN {X 0,Y 339.015,Z 472.339,A -85,B 0,C 180,E1 -14469.278,E2 -14469.278} C_VEL
LIN {X 0,Y 339.854,Z 483.35,A -85,B 0,C 180,E1 -14470.288,E2 -14470.288} C_VEL
LIN {X 0,Y 339.625,Z 490.156,A -85,B 0,C 180,E1 -14470.979,E2 -14470.979} C_VEL
LIN {X 0,Y 337.994,Z 501.626,A -85,B 0,C 180,E1 -14472.296,E2 -14472.296} C_VEL
LIN {X 0,Y 336.614,Z 511.34,A -85,B 0,C 180,E1 -14473.692,E2 -14473.692} C_VEL
LIN {X 0,Y 335.339,Z 521.042,A -85,B 0,C 180,E1 -14475.435,E2 -14475.435} C_VEL
LIN {X 0,Y 334.107,Z 529.189,A -85,B 0,C 180,E1 -14477.24,E2 -14477.24} C_VEL
LIN {X 0,Y 333.231,Z 535.776,A -85,B 0,C 180,E1 -14479.059,E2 -14479.059} C_VEL
LIN {X 0,Y 332.606,Z 541.038,A -85,B 0,C 180,E1 -14480.882,E2 -14480.882} C_VEL
LIN {X 0,Y 332.2,Z 545.146,A -85,B 0,C 180,E1 -14482.708,E2 -14482.708} C_VEL
LIN {X 0,Y 332.031,Z 547.66,A -85,B 0,C 180,E1 -14484.176,E2 -14484.176} C_VEL
LIN {X 0,Y 332,Z 550.294,A -85,B 0,C 180,E1 -14486.359,E2 -14486.359} C_VEL
LIN {X 0,Y 331.942,Z 551.183,A -85,B 0,C 180,E1 -14487.574,E2 -14487.574} C_VEL
LIN {X 0,Y 331.988,Z 551.637,A -85,B 0,C 180,E1 -14488.787,E2 -14488.787} C_VEL
LIN {X 0,Y 332.046,Z 551.698,A -85,B 0,C 180,E1 -14490,E2 -14490} C_VEL
LIN {X 0,Y 331.996,Z 551.362,A -85,B 0,C 180,E1 -14491.213,E2 -14491.213} C_VEL
LIN {X 0,Y 331.957,Z 550.618,A -85,B 0,C 180,E1 -14492.427,E2 -14492.427} C_VEL
LIN {X 0,Y 332.007,Z 549.425,A -85,B 0,C 180,E1 -14493.641,E2 -14493.641} C_VEL
LIN {X 0,Y 332.03,Z 546.227,A -85,B 0,C 180,E1 -14495.822,E2 -14495.822} C_VEL
LIN {X 0,Y 332.317,Z 541.809,A -85,B 0,C 180,E1 -14497.902,E2 -14497.902} C_VEL
LIN {X 0,Y 332.837,Z 535.674,A -85,B 0,C 180,E1 -14500.033,E2 -14500.033} C_VEL
LIN {X 0,Y 333.432,Z 528.949,A -85,B 0,C 180,E1 -14501.86,E2 -14501.86} C_VEL
LIN {X 0,Y 334.486,Z 520.62,A -85,B 0,C 180,E1 -14503.673,E2 -14503.673} C_VEL
LIN {X 0,Y 335.547,Z 510.867,A -85,B 0,C 180,E1 -14505.366,E2 -14505.366} C_VEL
LIN {X 0,Y 336.646,Z 500.32,A -85,B 0,C 180,E1 -14506.838,E2 -14506.838} C_VEL
LIN {X 0,Y 337.882,Z 489.659,A -85,B 0,C 180,E1 -14508.024,E2 -14508.024} C_VEL
LIN {X 0,Y 338.335,Z 484.956,A -85,B 0,C 180,E1 -14508.468,E2 -14508.468} C_VEL
LIN {X 0,Y 337.182,Z 472.247,A -85,B 0,C 180,E1 -14509.562,E2 -14509.562} C_VEL
LIN {X 0,Y 335.264,Z 458.835,A -85,B 0,C 180,E1 -14510.476,E2 -14510.476} C_VEL
LIN {X 0,Y 332.904,Z 445.341,A -85,B 0,C 180,E1 -14511.169,E2 -14511.169} C_VEL
LIN {X 0,Y 333.404,Z 438.763,A -85,B 0,C 180,E1 -14514.984,E2 -14514.984} C_VEL
LIN {X 0,Y 334.09,Z 432.099,A -85,B 0,C 180,E1 -14518.936,E2 -14518.936} C_VEL
LIN {X 0,Y 334.803,Z 425.608,A -85,B 0,C 180,E1 -14522.896,E2 -14522.896} C_VEL
LIN {X 0,Y 335.294,Z 421.976,A -85,B 0,C 180,E1 -14525.167,E2 -14525.167} C_VEL
LIN {X 0,Y 335.118,Z 417.353,A -85,B 0,C 180,E1 -14528.219,E2 -14528.219} C_VEL
LIN {X 0,Y 334.357,Z 412.655,A -85,B 0,C 180,E1 -14531.513,E2 -14531.513} C_VEL
LIN {X 0,Y 333.664,Z 408.924,A -85,B 0,C 180,E1 -14534.263,E2 -14534.263} C_VEL
LIN {X 0,Y 333.643,Z 408.924,A -85,B 0,C 180,E1 -14537.618,E2 -14537.618} C_VEL
LIN {X 0,Y 333.654,Z 408.926,A -85,B 0,C 180,E1 -14541.202,E2 -14541.202} C_VEL
LIN {X 0,Y 333.677,Z 408.918,A -85,B 0,C 180,E1 -14543.861,E2 -14543.861} C_VEL
LIN {X 0,Y 333.645,Z 408.925,A -85,B 0,C 180,E1 -14547.413,E2 -14547.413} C_VEL
LIN {X 0,Y 333.712,Z 408.918,A -85,B 0,C 180,E1 -14551.028,E2 -14551.028} C_VEL
LIN {X 0,Y 333.737,Z 408.911,A -85,B 0,C 180,E1 -14553.754,E2 -14553.754} C_VEL
LIN {X 0,Y 333.721,Z 408.912,A -85,B 0,C 180,E1 -14557.914,E2 -14557.914} C_VEL
LIN {X 0,Y 333.795,Z 408.904,A -85,B 0,C 180,E1 -14561.589,E2 -14561.589} C_VEL
LIN {X 0,Y 333.809,Z 408.902,A -85,B 0,C 180,E1 -14565.576,E2 -14565.576} C_VEL
LIN {X 0,Y 333.835,Z 408.903,A -85,B 0,C 180,E1 -14569.078,E2 -14569.078} C_VEL
LIN {X 0,Y 334.026,Z 408.878,A -85,B 0,C 180,E1 -14572.747,E2 -14572.747} C_VEL
LIN {X 0,Y 333.81,Z 408.905,A -85,B 0,C 180,E1 -14575.169,E2 -14575.169} C_VEL
LIN {X 0,Y 334.106,Z 408.865,A -85,B 0,C 180,E1 -14577.589,E2 -14577.589} C_VEL
LIN {X 0,Y 334.228,Z 408.849,A -85,B 0,C 180,E1 -14580,E2 -14580} C_VEL
LIN {X 0,Y 334.105,Z 408.866,A -85,B 0,C 180,E1 -14582.411,E2 -14582.411} C_VEL
LIN {X 0,Y 334.026,Z 408.877,A -85,B 0,C 180,E1 -14587.252,E2 -14587.252} C_VEL
LIN {X 0,Y 333.834,Z 408.904,A -85,B 0,C 180,E1 -14590.922,E2 -14590.922} C_VEL
LIN {X 0,Y 333.809,Z 408.905,A -85,B 0,C 180,E1 -14594.634,E2 -14594.634} C_VEL
LIN {X 0,Y 333.798,Z 408.907,A -85,B 0,C 180,E1 -14598.655,E2 -14598.655} C_VEL
LIN {X 0,Y 333.693,Z 408.917,A -85,B 0,C 180,E1 -14602.278,E2 -14602.278} C_VEL
LIN {X 0,Y 333.737,Z 408.912,A -85,B 0,C 180,E1 -14606.246,E2 -14606.246} C_VEL
LIN {X 0,Y 333.712,Z 408.917,A -85,B 0,C 180,E1 -14608.972,E2 -14608.972} C_VEL
LIN {X 0,Y 333.644,Z 408.926,A -85,B 0,C 180,E1 -14612.587,E2 -14612.587} C_VEL
LIN {X 0,Y 333.677,Z 408.919,A -85,B 0,C 180,E1 -14616.139,E2 -14616.139} C_VEL
LIN {X 0,Y 333.647,Z 408.923,A -85,B 0,C 180,E1 -14619.192,E2 -14619.192} C_VEL
LIN {X 0,Y 333.633,Z 408.928,A -85,B 0,C 180,E1 -14622.5,E2 -14622.5} C_VEL
LIN {X 0,Y 333.597,Z 408.928,A -85,B 0,C 180,E1 -14625.955,E2 -14625.955} C_VEL
LIN {X 0,Y 333.648,Z 408.922,A -85,B 0,C 180,E1 -14629.315,E2 -14629.315} C_VEL
LIN {X 0,Y 333.668,Z 408.92,A -85,B 0,C 180,E1 -14633.167,E2 -14633.167} C_VEL
LIN {X 0,Y 333.638,Z 408.926,A -85,B 0,C 180,E1 -14636.792,E2 -14636.792} C_VEL
LIN {X 0,Y 333.696,Z 408.915,A -85,B 0,C 180,E1 -14639.713,E2 -14639.713} C_VEL
LIN {X 0,Y 333.741,Z 408.915,A -85,B 0,C 180,E1 -14642.401,E2 -14642.401} C_VEL
LIN {X 0,Y 333.729,Z 408.912,A -85,B 0,C 180,E1 -14645.091,E2 -14645.091} C_VEL
LIN {X 0,Y 333.682,Z 408.918,A -85,B 0,C 180,E1 -14649.019,E2 -14649.019} C_VEL
LIN {X 0,Y 333.795,Z 408.903,A -85,B 0,C 180,E1 -14651.589,E2 -14651.589} C_VEL
LIN {X 0,Y 333.81,Z 408.901,A -85,B 0,C 180,E1 -14655.576,E2 -14655.576} C_VEL
LIN {X 0,Y 333.836,Z 408.898,A -85,B 0,C 180,E1 -14659.078,E2 -14659.078} C_VEL
LIN {X 0,Y 334.029,Z 408.876,A -85,B 0,C 180,E1 -14662.747,E2 -14662.747} C_VEL
LIN {X 0,Y 333.81,Z 408.901,A -85,B 0,C 180,E1 -14665.169,E2 -14665.169} C_VEL
LIN {X 0,Y 334.106,Z 408.865,A -85,B 0,C 180,E1 -14667.588,E2 -14667.588} C_VEL
LIN {X 0,Y 334.247,Z 408.85,A -85,B 0,C 180,E1 -14670,E2 -14670} C_VEL
LIN {X 0,Y 334.108,Z 408.869,A -85,B 0,C 180,E1 -14672.411,E2 -14672.411} C_VEL
LIN {X 0,Y 333.93,Z 408.89,A -85,B 0,C 180,E1 -14676.04,E2 -14676.04} C_VEL
LIN {X 0,Y 333.582,Z 408.934,A -85,B 0,C 180,E1 -14678.48,E2 -14678.48} C_VEL
LIN {X 0,Y 333.398,Z 409.233,A -85,B 0,C 180,E1 -14679.708,E2 -14679.708} C_VEL
LIN {X 0,Y 333.165,Z 413.584,A -85,B 0,C 180,E1 -14683.986,E2 -14683.986} C_VEL
LIN {X 0,Y 332.725,Z 418.268,A -85,B 0,C 180,E1 -14688.471,E2 -14688.471} C_VEL
LIN {X 0,Y 332.528,Z 421.997,A -85,B 0,C 180,E1 -14691.918,E2 -14691.918} C_VEL
LIN {X 0,Y 336.18,Z 437.18,A -85,B 0,C 180,E1 -14692.821,E2 -14692.821} C_VEL
LIN {X 0,Y 338.565,Z 448.955,A -85,B 0,C 180,E1 -14693.715,E2 -14693.715} C_VEL
LIN {X 0,Y 339.447,Z 454.09,A -85,B 0,C 180,E1 -14694.168,E2 -14694.168} C_VEL
LIN {X 0,Y 338.384,Z 465.441,A -85,B 0,C 180,E1 -14695.199,E2 -14695.199} C_VEL
LIN {X 0,Y 337.27,Z 476.929,A -85,B 0,C 180,E1 -14696.529,E2 -14696.529} C_VEL
LIN {X 0,Y 336.194,Z 486.406,A -85,B 0,C 180,E1 -14697.887,E2 -14697.887} C_VEL
LIN {X 0,Y 335.146,Z 495.636,A -85,B 0,C 180,E1 -14699.524,E2 -14699.524} C_VEL
LIN {X 0,Y 334.069,Z 504.236,A -85,B 0,C 180,E1 -14701.423,E2 -14701.423} C_VEL
LIN {X 0,Y 333.37,Z 510.782,A -85,B 0,C 180,E1 -14703.237,E2 -14703.237} C_VEL
LIN {X 0,Y 332.664,Z 517.098,A -85,B 0,C 180,E1 -14705.518,E2 -14705.518} C_VEL
LIN {X 0,Y 332.208,Z 521.756,A -85,B 0,C 180,E1 -14707.843,E2 -14707.843} C_VEL
LIN {X 0,Y 331.883,Z 524.881,A -85,B 0,C 180,E1 -14710.329,E2 -14710.329} C_VEL
LIN {X 0,Y 331.797,Z 526.281,A -85,B 0,C 180,E1 -14712.672,E2 -14712.672} C_VEL
LIN {X 0,Y 331.793,Z 526.347,A -85,B 0,C 180,E1 -14714.346,E2 -14714.346} C_VEL
LIN {X 0,Y 331.924,Z 525.636,A -85,B 0,C 180,E1 -14716.045,E2 -14716.045} C_VEL
LIN {X 0,Y 332.172,Z 524.118,A -85,B 0,C 180,E1 -14717.775,E2 -14717.775} C_VEL
LIN {X 0,Y 332.738,Z 520.707,A -85,B 0,C 180,E1 -14720.118,E2 -14720.118} C_VEL
LIN {X 0,Y 333.386,Z 515.969,A -85,B 0,C 180,E1 -14722.314,E2 -14722.314} C_VEL
LIN {X 0,Y 334.121,Z 511.459,A -85,B 0,C 180,E1 -14723.917,E2 -14723.917} C_VEL
LIN {X 0,Y 335.197,Z 504.565,A -85,B 0,C 180,E1 -14725.857,E2 -14725.857} C_VEL
LIN {X 0,Y 336.343,Z 497.036,A -85,B 0,C 180,E1 -14727.562,E2 -14727.562} C_VEL
LIN {X 0,Y 336.058,Z 494.579,A -85,B 0,C 180,E1 -14728.1,E2 -14728.1} C_VEL
LIN {X 0,Y 331.835,Z 486.757,A -85,B 0,C 180,E1 -14729.853,E2 -14729.853} C_VEL
LIN {X 0,Y 331.733,Z 483.896,A -85,B 0,C 180,E1 -14730.327,E2 -14730.327} C_VEL
LIN {X 0,Y 333.315,Z 473.018,A -85,B 0,C 180,E1 -14731.787,E2 -14731.787} C_VEL
LIN {X 0,Y 334.653,Z 461.907,A -85,B 0,C 180,E1 -14732.982,E2 -14732.982} C_VEL
LIN {X 0,Y 335.019,Z 457.956,A -85,B 0,C 180,E1 -14733.345,E2 -14733.345} C_VEL
LIN {X 0,Y 332.812,Z 446.252,A -85,B 0,C 180,E1 -14734.527,E2 -14734.527} C_VEL
LIN {X 0,Y 329.449,Z 434.185,A -85,B 0,C 180,E1 -14735.594,E2 -14735.594} C_VEL
LIN {X 0,Y 326.026,Z 424.203,A -85,B 0,C 180,E1 -14736.371,E2 -14736.371} C_VEL
LIN {X 0,Y 325.994,Z 423.848,A -85,B 0,C 180,E1 -14736.495,E2 -14736.495} C_VEL
LIN {X 0,Y 326.256,Z 420.743,A -85,B 0,C 180,E1 -14739.839,E2 -14739.839} C_VEL
LIN {X 0,Y 326.517,Z 418.389,A -85,B 0,C 180,E1 -14742.462,E2 -14742.462} C_VEL
LIN {X 0,Y 326.904,Z 415.066,A -85,B 0,C 180,E1 -14746.321,E2 -14746.321} C_VEL
LIN {X 0,Y 327.078,Z 412.041,A -85,B 0,C 180,E1 -14750.102,E2 -14750.102} C_VEL
LIN {X 0,Y 327.059,Z 410.211,A -85,B 0,C 180,E1 -14752.592,E2 -14752.592} C_VEL
LIN {X 0,Y 326.993,Z 409.755,A -85,B 0,C 180,E1 -14753.831,E2 -14753.831} C_VEL
LIN {X 0,Y 327.044,Z 409.75,A -85,B 0,C 180,E1 -14757.537,E2 -14757.537} C_VEL
LIN {X 0,Y 327.215,Z 409.728,A -85,B 0,C 180,E1 -14760,E2 -14760} C_VEL
LIN {X 0,Y 327.044,Z 409.746,A -85,B 0,C 180,E1 -14762.463,E2 -14762.463} C_VEL
LIN {X 0,Y 326.992,Z 409.755,A -85,B 0,C 180,E1 -14766.169,E2 -14766.169} C_VEL
LIN {X 0,Y 326.911,Z 409.765,A -85,B 0,C 180,E1 -14768.655,E2 -14768.655} C_VEL
LIN {X 0,Y 326.731,Z 409.788,A -85,B 0,C 180,E1 -14772.422,E2 -14772.422} C_VEL
LIN {X 0,Y 326.75,Z 409.785,A -85,B 0,C 180,E1 -14774.958,E2 -14774.958} C_VEL
LIN {X 0,Y 326.73,Z 409.787,A -85,B 0,C 180,E1 -14778.839,E2 -14778.839} C_VEL
LIN {X 0,Y 326.617,Z 409.802,A -85,B 0,C 180,E1 -14782.788,E2 -14782.788} C_VEL
LIN {X 0,Y 326.687,Z 409.794,A -85,B 0,C 180,E1 -14785.484,E2 -14785.484} C_VEL
LIN {X 0,Y 326.658,Z 409.797,A -85,B 0,C 180,E1 -14789.66,E2 -14789.66} C_VEL
LIN {X 0,Y 326.605,Z 409.806,A -85,B 0,C 180,E1 -14794.02,E2 -14794.02} C_VEL
LIN {X 0,Y 326.628,Z 409.803,A -85,B 0,C 180,E1 -14797.24,E2 -14797.24} C_VEL
LIN {X 0,Y 326.627,Z 409.946,A -85,B 0,C 180,E1 -14800.86,E2 -14800.86} C_VEL
LIN {X 0,Y 327.051,Z 412.284,A -85,B 0,C 180,E1 -14803.444,E2 -14803.444} C_VEL
LIN {X 0,Y 327.623,Z 415.739,A -85,B 0,C 180,E1 -14806.832,E2 -14806.832} C_VEL
LIN {X 0,Y 328.296,Z 419.821,A -85,B 0,C 180,E1 -14810.414,E2 -14810.414} C_VEL
LIN {X 0,Y 328.627,Z 422.124,A -85,B 0,C 180,E1 -14812.306,E2 -14812.306} C_VEL
LIN {X 0,Y 328.598,Z 425.358,A -85,B 0,C 180,E1 -14814.728,E2 -14814.728} C_VEL
LIN {X 0,Y 327.986,Z 429.489,A -85,B 0,C 180,E1 -14817.61,E2 -14817.61} C_VEL
LIN {X 0,Y 327.07,Z 435.821,A -85,B 0,C 180,E1 -14821.789,E2 -14821.789} C_VEL
LIN {X 0,Y 326.358,Z 442.277,A -85,B 0,C 180,E1 -14825.849,E2 -14825.849} C_VEL
LIN {X 0,Y 326.267,Z 443.523,A -85,B 0,C 180,E1 -14826.612,E2 -14826.612} C_VEL
LIN {X 0,Y 329.884,Z 458.373,A -85,B 0,C 180,E1 -14827.629,E2 -14827.629} C_VEL
LIN {X 0,Y 332.036,Z 470.818,A -85,B 0,C 180,E1 -14828.642,E2 -14828.642} C_VEL
LIN {X 0,Y 333.087,Z 482.548,A -85,B 0,C 180,E1 -14829.742,E2 -14829.742} C_VEL
LIN {X 0,Y 333.081,Z 489.147,A -85,B 0,C 180,E1 -14830.43,E2 -14830.43} C_VEL
LIN {X 0,Y 331.441,Z 500.734,A -85,B 0,C 180,E1 -14831.775,E2 -14831.775} C_VEL
LIN {X 0,Y 329.957,Z 510.454,A -85,B 0,C 180,E1 -14833.178,E2 -14833.178} C_VEL
LIN {X 0,Y 328.711,Z 519.683,A -85,B 0,C 180,E1 -14834.833,E2 -14834.833} C_VEL
LIN {X 0,Y 327.4,Z 527.927,A -85,B 0,C 180,E1 -14836.659,E2 -14836.659} C_VEL
LIN {X 0,Y 326.32,Z 534.673,A -85,B 0,C 180,E1 -14838.509,E2 -14838.509} C_VEL
LIN {X 0,Y 325.575,Z 540.906,A -85,B 0,C 180,E1 -14840.683,E2 -14840.683} C_VEL
LIN {X 0,Y 325.152,Z 544.982,A -85,B 0,C 180,E1 -14842.549,E2 -14842.549} C_VEL
LIN {X 0,Y 324.948,Z 547.711,A -85,B 0,C 180,E1 -14844.208,E2 -14844.208} C_VEL
LIN {X 0,Y 324.904,Z 550.075,A -85,B 0,C 180,E1 -14846.28,E2 -14846.28} C_VEL
LIN {X 0,Y 324.86,Z 550.934,A -85,B 0,C 180,E1 -14847.521,E2 -14847.521} C_VEL
LIN {X 0,Y 324.892,Z 551.369,A -85,B 0,C 180,E1 -14848.761,E2 -14848.761} C_VEL
LIN {X 0,Y 324.951,Z 551.414,A -85,B 0,C 180,E1 -14850,E2 -14850} C_VEL
LIN {X 0,Y 324.901,Z 551.062,A -85,B 0,C 180,E1 -14851.24,E2 -14851.24} C_VEL
LIN {X 0,Y 324.874,Z 550.286,A -85,B 0,C 180,E1 -14852.48,E2 -14852.48} C_VEL
LIN {X 0,Y 324.933,Z 549.074,A -85,B 0,C 180,E1 -14853.721,E2 -14853.721} C_VEL
LIN {X 0,Y 324.927,Z 546.171,A -85,B 0,C 180,E1 -14855.755,E2 -14855.755} C_VEL
LIN {X 0,Y 325.244,Z 541.378,A -85,B 0,C 180,E1 -14858.075,E2 -14858.075} C_VEL
LIN {X 0,Y 325.797,Z 535.179,A -85,B 0,C 180,E1 -14860.252,E2 -14860.252} C_VEL
LIN {X 0,Y 326.454,Z 528.403,A -85,B 0,C 180,E1 -14862.117,E2 -14862.117} C_VEL
LIN {X 0,Y 327.498,Z 519.999,A -85,B 0,C 180,E1 -14863.971,E2 -14863.971} C_VEL
LIN {X 0,Y 328.536,Z 511.143,A -85,B 0,C 180,E1 -14865.541,E2 -14865.541} C_VEL
LIN {X 0,Y 329.67,Z 500.687,A -85,B 0,C 180,E1 -14867.046,E2 -14867.046} C_VEL
LIN {X 0,Y 330.932,Z 490.186,A -85,B 0,C 180,E1 -14868.255,E2 -14868.255} C_VEL
LIN {X 0,Y 331.277,Z 483.866,A -85,B 0,C 180,E1 -14868.877,E2 -14868.877} C_VEL
LIN {X 0,Y 330.152,Z 472.062,A -85,B 0,C 180,E1 -14869.913,E2 -14869.913} C_VEL
LIN {X 0,Y 328.214,Z 458.678,A -85,B 0,C 180,E1 -14870.854,E2 -14870.854} C_VEL
LIN {X 0,Y 325.882,Z 445.107,A -85,B 0,C 180,E1 -14871.553,E2 -14871.553} C_VEL
LIN {X 0,Y 326.386,Z 438.481,A -85,B 0,C 180,E1 -14875.509,E2 -14875.509} C_VEL
LIN {X 0,Y 327.15,Z 431.736,A -85,B 0,C 180,E1 -14879.611,E2 -14879.611} C_VEL
LIN {X 0,Y 327.982,Z 424.983,A -85,B 0,C 180,E1 -14883.858,E2 -14883.858} C_VEL
LIN {X 0,Y 328.269,Z 422.347,A -85,B 0,C 180,E1 -14885.555,E2 -14885.555} C_VEL
LIN {X 0,Y 328.069,Z 418.139,A -85,B 0,C 180,E1 -14888.408,E2 -14888.408} C_VEL
LIN {X 0,Y 327.31,Z 413.493,A -85,B 0,C 180,E1 -14891.731,E2 -14891.731} C_VEL
LIN {X 0,Y 326.599,Z 409.803,A -85,B 0,C 180,E1 -14894.536,E2 -14894.536} C_VEL
LIN {X 0,Y 326.577,Z 409.802,A -85,B 0,C 180,E1 -14898.154,E2 -14898.154} C_VEL
LIN {X 0,Y 326.599,Z 409.803,A -85,B 0,C 180,E1 -14901.388,E2 -14901.388} C_VEL
LIN {X 0,Y 326.62,Z 409.799,A -85,B 0,C 180,E1 -14904.851,E2 -14904.851} C_VEL
LIN {X 0,Y 326.609,Z 409.801,A -85,B 0,C 180,E1 -14907.455,E2 -14907.455} C_VEL
LIN {X 0,Y 326.662,Z 409.792,A -85,B 0,C 180,E1 -14910.341,E2 -14910.341} C_VEL
LIN {X 0,Y 326.691,Z 409.788,A -85,B 0,C 180,E1 -14914.516,E2 -14914.516} C_VEL
LIN {X 0,Y 326.647,Z 409.794,A -85,B 0,C 180,E1 -14918.545,E2 -14918.545} C_VEL
LIN {X 0,Y 326.746,Z 409.786,A -85,B 0,C 180,E1 -14921.177,E2 -14921.177} C_VEL
LIN {X 0,Y 326.764,Z 409.781,A -85,B 0,C 180,E1 -14925.433,E2 -14925.433} C_VEL
LIN {X 0,Y 326.771,Z 409.782,A -85,B 0,C 180,E1 -14928.839,E2 -14928.839} C_VEL
LIN {X 0,Y 326.98,Z 409.754,A -85,B 0,C 180,E1 -14932.59,E2 -14932.59} C_VEL
LIN {X 0,Y 326.778,Z 409.782,A -85,B 0,C 180,E1 -14935.065,E2 -14935.065} C_VEL
LIN {X 0,Y 327.046,Z 409.744,A -85,B 0,C 180,E1 -14937.537,E2 -14937.537} C_VEL
LIN {X 0,Y 327.18,Z 409.727,A -85,B 0,C 180,E1 -14940,E2 -14940} C_VEL
LIN {X 0,Y 327.046,Z 409.745,A -85,B 0,C 180,E1 -14942.463,E2 -14942.463} C_VEL
LIN {X 0,Y 326.972,Z 409.751,A -85,B 0,C 180,E1 -14946.656,E2 -14946.656} C_VEL
LIN {X 0,Y 326.814,Z 409.772,A -85,B 0,C 180,E1 -14949.906,E2 -14949.906} C_VEL
LIN {X 0,Y 326.76,Z 409.779,A -85,B 0,C 180,E1 -14953.685,E2 -14953.685} C_VEL
LIN {X 0,Y 326.7,Z 409.787,A -85,B 0,C 180,E1 -14957.528,E2 -14957.528} C_VEL
LIN {X 0,Y 326.666,Z 409.791,A -85,B 0,C 180,E1 -14960.135,E2 -14960.135} C_VEL
LIN {X 0,Y 326.653,Z 409.793,A -85,B 0,C 180,E1 -14964.129,E2 -14964.129} C_VEL
LIN {X 0,Y 326.686,Z 409.793,A -85,B 0,C 180,E1 -14966.858,E2 -14966.858} C_VEL
LIN {X 0,Y 326.64,Z 409.799,A -85,B 0,C 180,E1 -14970.611,E2 -14970.611} C_VEL
LIN {X 0,Y 326.608,Z 409.799,A -85,B 0,C 180,E1 -14974.019,E2 -14974.019} C_VEL
LIN {X 0,Y 326.628,Z 409.797,A -85,B 0,C 180,E1 -14977.238,E2 -14977.238} C_VEL
LIN {X 0,Y 326.578,Z 409.803,A -85,B 0,C 180,E1 -14981.131,E2 -14981.131} C_VEL
LIN {X 0,Y 326.528,Z 409.813,A -85,B 0,C 180,E1 -14984.743,E2 -14984.743} C_VEL
LIN {X 0,Y 326.577,Z 409.804,A -85,B 0,C 180,E1 -14988.154,E2 -14988.154} C_VEL
LIN {X 0,Y 326.626,Z 409.796,A -85,B 0,C 180,E1 -14991.391,E2 -14991.391} C_VEL
LIN {X 0,Y 326.621,Z 409.799,A -85,B 0,C 180,E1 -14994.851,E2 -14994.851} C_VEL
LIN {X 0,Y 326.609,Z 409.798,A -85,B 0,C 180,E1 -14997.455,E2 -14997.455} C_VEL
LIN {X 0,Y 326.649,Z 409.797,A -85,B 0,C 180,E1 -15000.34,E2 -15000.34} C_VEL
LIN {X 0,Y 326.692,Z 409.793,A -85,B 0,C 180,E1 -15004.516,E2 -15004.516} C_VEL
LIN {X 0,Y 326.647,Z 409.798,A -85,B 0,C 180,E1 -15008.545,E2 -15008.545} C_VEL
LIN {X 0,Y 326.746,Z 409.781,A -85,B 0,C 180,E1 -15011.177,E2 -15011.177} C_VEL
LIN {X 0,Y 326.765,Z 409.778,A -85,B 0,C 180,E1 -15015.433,E2 -15015.433} C_VEL
LIN {X 0,Y 326.772,Z 409.779,A -85,B 0,C 180,E1 -15018.839,E2 -15018.839} C_VEL
LIN {X 0,Y 326.98,Z 409.755,A -85,B 0,C 180,E1 -15022.59,E2 -15022.59} C_VEL
LIN {X 0,Y 326.778,Z 409.777,A -85,B 0,C 180,E1 -15025.064,E2 -15025.064} C_VEL
LIN {X 0,Y 327.047,Z 409.744,A -85,B 0,C 180,E1 -15027.536,E2 -15027.536} C_VEL
LIN {X 0,Y 327.199,Z 409.727,A -85,B 0,C 180,E1 -15030,E2 -15030} C_VEL
LIN {X 0,Y 327.048,Z 409.747,A -85,B 0,C 180,E1 -15032.463,E2 -15032.463} C_VEL
LIN {X 0,Y 326.877,Z 409.77,A -85,B 0,C 180,E1 -15036.171,E2 -15036.171} C_VEL
LIN {X 0,Y 326.512,Z 409.813,A -85,B 0,C 180,E1 -15038.665,E2 -15038.665} C_VEL
LIN {X 0,Y 326.327,Z 410.324,A -85,B 0,C 180,E1 -15039.921,E2 -15039.921} C_VEL
LIN {X 0,Y 326.083,Z 414.497,A -85,B 0,C 180,E1 -15044.099,E2 -15044.099} C_VEL
LIN {X 0,Y 325.683,Z 418.857,A -85,B 0,C 180,E1 -15048.288,E2 -15048.288} C_VEL
LIN {X 0,Y 325.478,Z 422.39,A -85,B 0,C 180,E1 -15051.535,E2 -15051.535} C_VEL
LIN {X 0,Y 328.778,Z 435.768,A -85,B 0,C 180,E1 -15052.329,E2 -15052.329} C_VEL
LIN {X 0,Y 331.296,Z 447.793,A -85,B 0,C 180,E1 -15053.245,E2 -15053.245} C_VEL
LIN {X 0,Y 332.49,Z 454.507,A -85,B 0,C 180,E1 -15053.844,E2 -15053.844} C_VEL
LIN {X 0,Y 331.512,Z 465.937,A -85,B 0,C 180,E1 -15054.914,E2 -15054.914} C_VEL
LIN {X 0,Y 330.429,Z 476.747,A -85,B 0,C 180,E1 -15056.189,E2 -15056.189} C_VEL
LIN {X 0,Y 329.242,Z 486.864,A -85,B 0,C 180,E1 -15057.662,E2 -15057.662} C_VEL
LIN {X 0,Y 328.175,Z 495.86,A -85,B 0,C 180,E1 -15059.293,E2 -15059.293} C_VEL
LIN {X 0,Y 327.189,Z 503.654,A -85,B 0,C 180,E1 -15061.031,E2 -15061.031} C_VEL
LIN {X 0,Y 326.399,Z 510.37,A -85,B 0,C 180,E1 -15062.887,E2 -15062.887} C_VEL
LIN {X 0,Y 325.728,Z 516.199,A -85,B 0,C 180,E1 -15064.925,E2 -15064.925} C_VEL
LIN {X 0,Y 325.221,Z 521.057,A -85,B 0,C 180,E1 -15067.234,E2 -15067.234} C_VEL
LIN {X 0,Y 324.966,Z 523.566,A -85,B 0,C 180,E1 -15068.87,E2 -15068.87} C_VEL
LIN {X 0,Y 324.753,Z 525.528,A -85,B 0,C 180,E1 -15070.761,E2 -15070.761} C_VEL
LIN {X 0,Y 324.702,Z 526.529,A -85,B 0,C 180,E1 -15072.616,E2 -15072.616} C_VEL
LIN {X 0,Y 324.701,Z 526.628,A -85,B 0,C 180,E1 -15074.417,E2 -15074.417} C_VEL
LIN {X 0,Y 324.844,Z 525.909,A -85,B 0,C 180,E1 -15076.186,E2 -15076.186} C_VEL
LIN {X 0,Y 325.108,Z 524.421,A -85,B 0,C 180,E1 -15077.922,E2 -15077.922} C_VEL
LIN {X 0,Y 325.728,Z 520.989,A -85,B 0,C 180,E1 -15080.335,E2 -15080.335} C_VEL
LIN {X 0,Y 326.247,Z 517.417,A -85,B 0,C 180,E1 -15082.089,E2 -15082.089} C_VEL
LIN {X 0,Y 327.176,Z 511.891,A -85,B 0,C 180,E1 -15084.172,E2 -15084.172} C_VEL
LIN {X 0,Y 328.327,Z 504.938,A -85,B 0,C 180,E1 -15086.183,E2 -15086.183} C_VEL
LIN {X 0,Y 329.715,Z 496.342,A -85,B 0,C 180,E1 -15088.15,E2 -15088.15} C_VEL
LIN {X 0,Y 331.306,Z 486.729,A -85,B 0,C 180,E1 -15089.879,E2 -15089.879} C_VEL
LIN {X 0,Y 331.733,Z 483.896,A -85,B 0,C 180,E1 -15090.327,E2 -15090.327} C_VEL
LIN {X 0,Y 332.063,Z 479.458,A -85,B 0,C 180,E1 -15090.991,E2 -15090.991} C_VEL
LIN {X 0,Y 330.847,Z 472.103,A -85,B 0,C 180,E1 -15092.103,E2 -15092.103} C_VEL
LIN {X 0,Y 328.734,Z 462.876,A -85,B 0,C 180,E1 -15093.366,E2 -15093.366} C_VEL
LIN {X 0,Y 328.359,Z 459.556,A -85,B 0,C 180,E1 -15093.74,E2 -15093.74} C_VEL
LIN {X 0,Y 326.572,Z 449.094,A -85,B 0,C 180,E1 -15094.847,E2 -15094.847} C_VEL
LIN {X 0,Y 323.447,Z 437.307,A -85,B 0,C 180,E1 -15095.964,E2 -15095.964} C_VEL
LIN {X 0,Y 319.483,Z 426.246,A -85,B 0,C 180,E1 -15096.922,E2 -15096.922} C_VEL
LIN {X 0,Y 318.967,Z 424.255,A -85,B 0,C 180,E1 -15097.089,E2 -15097.089} C_VEL
LIN {X 0,Y 319.375,Z 420.617,A -85,B 0,C 180,E1 -15101.124,E2 -15101.124} C_VEL
LIN {X 0,Y 319.813,Z 417.113,A -85,B 0,C 180,E1 -15105.217,E2 -15105.217} C_VEL
LIN {X 0,Y 320.028,Z 414.406,A -85,B 0,C 180,E1 -15108.601,E2 -15108.601} C_VEL
LIN {X 0,Y 320.1,Z 412.496,A -85,B 0,C 180,E1 -15111.159,E2 -15111.159} C_VEL
LIN {X 0,Y 319.978,Z 410.746,A -85,B 0,C 180,E1 -15113.695,E2 -15113.695} C_VEL
LIN {X 0,Y 319.988,Z 410.629,A -85,B 0,C 180,E1 -15117.482,E2 -15117.482} C_VEL
LIN {X 0,Y 320.166,Z 410.605,A -85,B 0,C 180,E1 -15120,E2 -15120} C_VEL
LIN {X 0,Y 319.988,Z 410.625,A -85,B 0,C 180,E1 -15122.518,E2 -15122.518} C_VEL
LIN {X 0,Y 319.948,Z 410.633,A -85,B 0,C 180,E1 -15126.306,E2 -15126.306} C_VEL
LIN {X 0,Y 319.839,Z 410.647,A -85,B 0,C 180,E1 -15128.848,E2 -15128.848} C_VEL
LIN {X 0,Y 319.678,Z 410.667,A -85,B 0,C 180,E1 -15132.7,E2 -15132.7} C_VEL
LIN {X 0,Y 319.696,Z 410.665,A -85,B 0,C 180,E1 -15135.296,E2 -15135.296} C_VEL
LIN {X 0,Y 319.671,Z 410.667,A -85,B 0,C 180,E1 -15139.255,E2 -15139.255} C_VEL
LIN {X 0,Y 319.567,Z 410.68,A -85,B 0,C 180,E1 -15143.32,E2 -15143.32} C_VEL
LIN {X 0,Y 319.632,Z 410.671,A -85,B 0,C 180,E1 -15146.088,E2 -15146.088} C_VEL
LIN {X 0,Y 319.587,Z 410.678,A -85,B 0,C 180,E1 -15148.934,E2 -15148.934} C_VEL
LIN {X 0,Y 319.531,Z 410.685,A -85,B 0,C 180,E1 -15151.862,E2 -15151.862} C_VEL
LIN {X 0,Y 319.578,Z 410.68,A -85,B 0,C 180,E1 -15155.544,E2 -15155.544} C_VEL
LIN {X 0,Y 319.596,Z 410.68,A -85,B 0,C 180,E1 -15158.005,E2 -15158.005} C_VEL
LIN {X 0,Y 319.597,Z 410.819,A -85,B 0,C 180,E1 -15160.031,E2 -15160.031} C_VEL
LIN {X 0,Y 320.142,Z 413.918,A -85,B 0,C 180,E1 -15163.579,E2 -15163.579} C_VEL
LIN {X 0,Y 320.732,Z 417.569,A -85,B 0,C 180,E1 -15167.213,E2 -15167.213} C_VEL
LIN {X 0,Y 321.368,Z 421.401,A -85,B 0,C 180,E1 -15170.64,E2 -15170.64} C_VEL
LIN {X 0,Y 321.647,Z 423.378,A -85,B 0,C 180,E1 -15172.281,E2 -15172.281} C_VEL
LIN {X 0,Y 321.648,Z 425.495,A -85,B 0,C 180,E1 -15173.945,E2 -15173.945} C_VEL
LIN {X 0,Y 321.117,Z 429.456,A -85,B 0,C 180,E1 -15176.829,E2 -15176.829} C_VEL
LIN {X 0,Y 320.255,Z 434.692,A -85,B 0,C 180,E1 -15180.413,E2 -15180.413} C_VEL
LIN {X 0,Y 319.55,Z 440.764,A -85,B 0,C 180,E1 -15184.387,E2 -15184.387} C_VEL
LIN {X 0,Y 319.283,Z 443.304,A -85,B 0,C 180,E1 -15185.971,E2 -15185.971} C_VEL
LIN {X 0,Y 322.949,Z 457.443,A -85,B 0,C 180,E1 -15186.974,E2 -15186.974} C_VEL
LIN {X 0,Y 325.233,Z 470.373,A -85,B 0,C 180,E1 -15188.057,E2 -15188.057} C_VEL
LIN {X 0,Y 326.366,Z 481.947,A -85,B 0,C 180,E1 -15189.184,E2 -15189.184} C_VEL
LIN {X 0,Y 326.421,Z 489.563,A -85,B 0,C 180,E1 -15190.014,E2 -15190.014} C_VEL
LIN {X 0,Y 324.724,Z 501.006,A -85,B 0,C 180,E1 -15191.384,E2 -15191.384} C_VEL
LIN {X 0,Y 323.165,Z 510.633,A -85,B 0,C 180,E1 -15192.814,E2 -15192.814} C_VEL
LIN {X 0,Y 321.823,Z 519.881,A -85,B 0,C 180,E1 -15194.528,E2 -15194.528} C_VEL
LIN {X 0,Y 320.47,Z 527.941,A -85,B 0,C 180,E1 -15196.365,E2 -15196.365} C_VEL
LIN {X 0,Y 319.336,Z 534.636,A -85,B 0,C 180,E1 -15198.254,E2 -15198.254} C_VEL
LIN {X 0,Y 318.541,Z 540.79,A -85,B 0,C 180,E1 -15200.476,E2 -15200.476} C_VEL
LIN {X 0,Y 318.076,Z 544.819,A -85,B 0,C 180,E1 -15202.382,E2 -15202.382} C_VEL
LIN {X 0,Y 317.841,Z 547.814,A -85,B 0,C 180,E1 -15204.286,E2 -15204.286} C_VEL
LIN {X 0,Y 317.811,Z 549.856,A -85,B 0,C 180,E1 -15206.197,E2 -15206.197} C_VEL
LIN {X 0,Y 317.78,Z 550.682,A -85,B 0,C 180,E1 -15207.465,E2 -15207.465} C_VEL
LIN {X 0,Y 317.8,Z 551.102,A -85,B 0,C 180,E1 -15208.733,E2 -15208.733} C_VEL
LIN {X 0,Y 317.856,Z 551.131,A -85,B 0,C 180,E1 -15210,E2 -15210} C_VEL
LIN {X 0,Y 317.808,Z 550.761,A -85,B 0,C 180,E1 -15211.268,E2 -15211.268} C_VEL
LIN {X 0,Y 317.795,Z 549.951,A -85,B 0,C 180,E1 -15212.535,E2 -15212.535} C_VEL
LIN {X 0,Y 317.838,Z 548.721,A -85,B 0,C 180,E1 -15213.804,E2 -15213.804} C_VEL
LIN {X 0,Y 317.848,Z 546.044,A -85,B 0,C 180,E1 -15215.728,E2 -15215.728} C_VEL
LIN {X 0,Y 318.069,Z 542.385,A -85,B 0,C 180,E1 -15217.619,E2 -15217.619} C_VEL
LIN {X 0,Y 318.476,Z 537.56,A -85,B 0,C 180,E1 -15219.527,E2 -15219.527} C_VEL
LIN {X 0,Y 319.041,Z 531.447,A -85,B 0,C 180,E1 -15221.435,E2 -15221.435} C_VEL
LIN {X 0,Y 320.036,Z 523.854,A -85,B 0,C 180,E1 -15223.332,E2 -15223.332} C_VEL
LIN {X 0,Y 321.015,Z 516.089,A -85,B 0,C 180,E1 -15224.907,E2 -15224.907} C_VEL
LIN {X 0,Y 322.084,Z 506.607,A -85,B 0,C 180,E1 -15226.479,E2 -15226.479} C_VEL
LIN {X 0,Y 323.321,Z 496.137,A -85,B 0,C 180,E1 -15227.881,E2 -15227.881} C_VEL
LIN {X 0,Y 324.438,Z 486.132,A -85,B 0,C 180,E1 -15228.962,E2 -15228.962} C_VEL
LIN {X 0,Y 323.469,Z 474.515,A -85,B 0,C 180,E1 -15230.064,E2 -15230.064} C_VEL
LIN {X 0,Y 321.664,Z 461.289,A -85,B 0,C 180,E1 -15231.063,E2 -15231.063} C_VEL
LIN {X 0,Y 319.415,Z 448.263,A -85,B 0,C 180,E1 -15231.815,E2 -15231.815} C_VEL
LIN {X 0,Y 318.876,Z 444.824,A -85,B 0,C 180,E1 -15232.005,E2 -15232.005} C_VEL
LIN {X 0,Y 319.411,Z 438.111,A -85,B 0,C 180,E1 -15236.108,E2 -15236.108} C_VEL
LIN {X 0,Y 320.076,Z 432.508,A -85,B 0,C 180,E1 -15239.607,E2 -15239.607} C_VEL
LIN {X 0,Y 320.876,Z 426.18,A -85,B 0,C 180,E1 -15243.664,E2 -15243.664} C_VEL
LIN {X 0,Y 321.21,Z 422.344,A -85,B 0,C 180,E1 -15246.211,E2 -15246.211} C_VEL
LIN {X 0,Y 321.001,Z 418.837,A -85,B 0,C 180,E1 -15248.655,E2 -15248.655} C_VEL
LIN {X 0,Y 320.311,Z 414.613,A -85,B 0,C 180,E1 -15251.755,E2 -15251.755} C_VEL
LIN {X 0,Y 319.521,Z 410.686,A -85,B 0,C 180,E1 -15254.837,E2 -15254.837} C_VEL
LIN {X 0,Y 319.527,Z 410.681,A -85,B 0,C 180,E1 -15258.403,E2 -15258.403} C_VEL
LIN {X 0,Y 319.544,Z 410.678,A -85,B 0,C 180,E1 -15261.988,E2 -15261.988} C_VEL
LIN {X 0,Y 319.562,Z 410.68,A -85,B 0,C 180,E1 -15265.123,E2 -15265.123} C_VEL
LIN {X 0,Y 319.572,Z 410.679,A -85,B 0,C 180,E1 -15269.058,E2 -15269.058} C_VEL
LIN {X 0,Y 319.609,Z 410.67,A -85,B 0,C 180,E1 -15272.498,E2 -15272.498} C_VEL
LIN {X 0,Y 319.607,Z 410.674,A -85,B 0,C 180,E1 -15275.304,E2 -15275.304} C_VEL
LIN {X 0,Y 319.598,Z 410.671,A -85,B 0,C 180,E1 -15278.048,E2 -15278.048} C_VEL
LIN {X 0,Y 319.69,Z 410.664,A -85,B 0,C 180,E1 -15280.962,E2 -15280.962} C_VEL
LIN {X 0,Y 319.732,Z 410.658,A -85,B 0,C 180,E1 -15285.276,E2 -15285.276} C_VEL
LIN {X 0,Y 319.759,Z 410.651,A -85,B 0,C 180,E1 -15289.873,E2 -15289.873} C_VEL
LIN {X 0,Y 319.934,Z 410.63,A -85,B 0,C 180,E1 -15292.426,E2 -15292.426} C_VEL
LIN {X 0,Y 319.747,Z 410.658,A -85,B 0,C 180,E1 -15294.956,E2 -15294.956} C_VEL
LIN {X 0,Y 319.99,Z 410.624,A -85,B 0,C 180,E1 -15297.482,E2 -15297.482} C_VEL
LIN {X 0,Y 320.132,Z 410.605,A -85,B 0,C 180,E1 -15300,E2 -15300} C_VEL
LIN {X 0,Y 319.99,Z 410.624,A -85,B 0,C 180,E1 -15302.518,E2 -15302.518} C_VEL
LIN {X 0,Y 319.932,Z 410.628,A -85,B 0,C 180,E1 -15306.647,E2 -15306.647} C_VEL
LIN {X 0,Y 319.759,Z 410.652,A -85,B 0,C 180,E1 -15310.127,E2 -15310.127} C_VEL
LIN {X 0,Y 319.732,Z 410.659,A -85,B 0,C 180,E1 -15314.724,E2 -15314.724} C_VEL
LIN {X 0,Y 319.69,Z 410.662,A -85,B 0,C 180,E1 -15319.038,E2 -15319.038} C_VEL
LIN {X 0,Y 319.571,Z 410.676,A -85,B 0,C 180,E1 -15323.319,E2 -15323.319} C_VEL
LIN {X 0,Y 319.636,Z 410.667,A -85,B 0,C 180,E1 -15326.088,E2 -15326.088} C_VEL
LIN {X 0,Y 319.591,Z 410.676,A -85,B 0,C 180,E1 -15328.933,E2 -15328.933} C_VEL
LIN {X 0,Y 319.533,Z 410.679,A -85,B 0,C 180,E1 -15331.862,E2 -15331.862} C_VEL
LIN {X 0,Y 319.58,Z 410.672,A -85,B 0,C 180,E1 -15335.543,E2 -15335.543} C_VEL
LIN {X 0,Y 319.558,Z 410.676,A -85,B 0,C 180,E1 -15338.01,E2 -15338.01} C_VEL
LIN {X 0,Y 319.526,Z 410.68,A -85,B 0,C 180,E1 -15341.597,E2 -15341.597} C_VEL
LIN {X 0,Y 319.489,Z 410.686,A -85,B 0,C 180,E1 -15345.257,E2 -15345.257} C_VEL
LIN {X 0,Y 319.53,Z 410.684,A -85,B 0,C 180,E1 -15348.712,E2 -15348.712} C_VEL
LIN {X 0,Y 319.58,Z 410.676,A -85,B 0,C 180,E1 -15352.344,E2 -15352.344} C_VEL
LIN {X 0,Y 319.562,Z 410.677,A -85,B 0,C 180,E1 -15355.123,E2 -15355.123} C_VEL
LIN {X 0,Y 319.568,Z 410.676,A -85,B 0,C 180,E1 -15359.059,E2 -15359.059} C_VEL
LIN {X 0,Y 319.608,Z 410.675,A -85,B 0,C 180,E1 -15362.498,E2 -15362.498} C_VEL
LIN {X 0,Y 319.607,Z 410.67,A -85,B 0,C 180,E1 -15365.304,E2 -15365.304} C_VEL
LIN {X 0,Y 319.598,Z 410.673,A -85,B 0,C 180,E1 -15368.048,E2 -15368.048} C_VEL
LIN {X 0,Y 319.691,Z 410.661,A -85,B 0,C 180,E1 -15370.962,E2 -15370.962} C_VEL
LIN {X 0,Y 319.733,Z 410.655,A -85,B 0,C 180,E1 -15375.275,E2 -15375.275} C_VEL
LIN {X 0,Y 319.76,Z 410.652,A -85,B 0,C 180,E1 -15379.873,E2 -15379.873} C_VEL
LIN {X 0,Y 319.936,Z 410.634,A -85,B 0,C 180,E1 -15382.426,E2 -15382.426} C_VEL
LIN {X 0,Y 319.748,Z 410.653,A -85,B 0,C 180,E1 -15384.956,E2 -15384.956} C_VEL
LIN {X 0,Y 319.991,Z 410.622,A -85,B 0,C 180,E1 -15387.482,E2 -15387.482} C_VEL
LIN {X 0,Y 320.151,Z 410.606,A -85,B 0,C 180,E1 -15390,E2 -15390} C_VEL
LIN {X 0,Y 319.992,Z 410.626,A -85,B 0,C 180,E1 -15392.517,E2 -15392.517} C_VEL
LIN {X 0,Y 319.806,Z 410.651,A -85,B 0,C 180,E1 -15396.308,E2 -15396.308} C_VEL
LIN {X 0,Y 319.424,Z 410.695,A -85,B 0,C 180,E1 -15398.859,E2 -15398.859} C_VEL
LIN {X 0,Y 319.246,Z 411.415,A -85,B 0,C 180,E1 -15400.143,E2 -15400.143} C_VEL
LIN {X 0,Y 319.015,Z 415.419,A -85,B 0,C 180,E1 -15404.226,E2 -15404.226} C_VEL
LIN {X 0,Y 318.601,Z 419.769,A -85,B 0,C 180,E1 -15408.462,E2 -15408.462} C_VEL
LIN {X 0,Y 318.445,Z 422.545,A -85,B 0,C 180,E1 -15411.1,E2 -15411.1} C_VEL
LIN {X 0,Y 322.231,Z 438.151,A -85,B 0,C 180,E1 -15412.082,E2 -15412.082} C_VEL
LIN {X 0,Y 324.587,Z 449.585,A -85,B 0,C 180,E1 -15413.006,E2 -15413.006} C_VEL
LIN {X 0,Y 325.636,Z 456.447,A -85,B 0,C 180,E1 -15413.652,E2 -15413.652} C_VEL
LIN {X 0,Y 324.499,Z 467.986,A -85,B 0,C 180,E1 -15414.788,E2 -15414.788} C_VEL
LIN {X 0,Y 323.357,Z 478.537,A -85,B 0,C 180,E1 -15416.095,E2 -15416.095} C_VEL
LIN {X 0,Y 322.106,Z 488.453,A -85,B 0,C 180,E1 -15417.622,E2 -15417.622} C_VEL
LIN {X 0,Y 321.126,Z 496.837,A -85,B 0,C 180,E1 -15419.212,E2 -15419.212} C_VEL
LIN {X 0,Y 320.061,Z 504.91,A -85,B 0,C 180,E1 -15421.088,E2 -15421.088} C_VEL
LIN {X 0,Y 319.305,Z 511.057,A -85,B 0,C 180,E1 -15422.862,E2 -15422.862} C_VEL
LIN {X 0,Y 318.625,Z 516.883,A -85,B 0,C 180,E1 -15424.993,E2 -15424.993} C_VEL
LIN {X 0,Y 318.11,Z 521.567,A -85,B 0,C 180,E1 -15427.312,E2 -15427.312} C_VEL
LIN {X 0,Y 317.798,Z 524.356,A -85,B 0,C 180,E1 -15429.284,E2 -15429.284} C_VEL
LIN {X 0,Y 317.623,Z 526.341,A -85,B 0,C 180,E1 -15431.59,E2 -15431.59} C_VEL
LIN {X 0,Y 317.612,Z 526.916,A -85,B 0,C 180,E1 -15433.31,E2 -15433.31} C_VEL
LIN {X 0,Y 317.64,Z 526.768,A -85,B 0,C 180,E1 -15435.073,E2 -15435.073} C_VEL
LIN {X 0,Y 317.832,Z 525.847,A -85,B 0,C 180,E1 -15436.861,E2 -15436.861} C_VEL
LIN {X 0,Y 318.383,Z 523.024,A -85,B 0,C 180,E1 -15439.455,E2 -15439.455} C_VEL
LIN {X 0,Y 318.882,Z 520.08,A -85,B 0,C 180,E1 -15441.223,E2 -15441.223} C_VEL
LIN {X 0,Y 319.554,Z 516.176,A -85,B 0,C 180,E1 -15443.012,E2 -15443.012} C_VEL
LIN {X 0,Y 320.653,Z 509.789,A -85,B 0,C 180,E1 -15445.259,E2 -15445.259} C_VEL
LIN {X 0,Y 321.967,Z 502.47,A -85,B 0,C 180,E1 -15447.243,E2 -15447.243} C_VEL
LIN {X 0,Y 323.49,Z 493.747,A -85,B 0,C 180,E1 -15449.119,E2 -15449.119} C_VEL
LIN {X 0,Y 325.019,Z 484.576,A -85,B 0,C 180,E1 -15450.71,E2 -15450.71} C_VEL
LIN {X 0,Y 326.717,Z 473.571,A -85,B 0,C 180,E1 -15452.23,E2 -15452.23} C_VEL
LIN {X 0,Y 328.154,Z 462.405,A -85,B 0,C 180,E1 -15453.461,E2 -15453.461} C_VEL
LIN {X 0,Y 328.359,Z 459.556,A -85,B 0,C 180,E1 -15453.74,E2 -15453.74} C_VEL
LIN {X 0,Y 327.816,Z 456.301,A -85,B 0,C 180,E1 -15454.111,E2 -15454.111} C_VEL
LIN {X 0,Y 326.599,Z 453.267,A -85,B 0,C 180,E1 -15454.494,E2 -15454.494} C_VEL
LIN {X 0,Y 323.171,Z 447.676,A -85,B 0,C 180,E1 -15455.284,E2 -15455.284} C_VEL
LIN {X 0,Y 319.246,Z 442.125,A -85,B 0,C 180,E1 -15456.066,E2 -15456.066} C_VEL
LIN {X 0,Y 316.709,Z 437.571,A -85,B 0,C 180,E1 -15456.613,E2 -15456.613} C_VEL
LIN {X 0,Y 316.041,Z 435.92,A -85,B 0,C 180,E1 -15456.781,E2 -15456.781} C_VEL
LIN {X 0,Y 312.041,Z 424.923,A -85,B 0,C 180,E1 -15457.752,E2 -15457.752} C_VEL
LIN {X 0,Y 312.012,Z 424.55,A -85,B 0,C 180,E1 -15457.834,E2 -15457.834} C_VEL
LIN {X 0,Y 312.397,Z 421.227,A -85,B 0,C 180,E1 -15461.642,E2 -15461.642} C_VEL
LIN {X 0,Y 312.847,Z 417.87,A -85,B 0,C 180,E1 -15465.693,E2 -15465.693} C_VEL
LIN {X 0,Y 313.067,Z 414.837,A -85,B 0,C 180,E1 -15469.654,E2 -15469.654} C_VEL
LIN {X 0,Y 313.105,Z 412.991,A -85,B 0,C 180,E1 -15472.26,E2 -15472.26} C_VEL
LIN {X 0,Y 313.004,Z 412.152,A -85,B 0,C 180,E1 -15473.554,E2 -15473.554} C_VEL
LIN {X 0,Y 312.717,Z 411.533,A -85,B 0,C 180,E1 -15474.842,E2 -15474.842} C_VEL
LIN {X 0,Y 312.989,Z 411.499,A -85,B 0,C 180,E1 -15478.713,E2 -15478.713} C_VEL
LIN {X 0,Y 313.118,Z 411.483,A -85,B 0,C 180,E1 -15480,E2 -15480} C_VEL
LIN {X 0,Y 312.934,Z 411.504,A -85,B 0,C 180,E1 -15482.575,E2 -15482.575} C_VEL
LIN {X 0,Y 312.906,Z 411.51,A -85,B 0,C 180,E1 -15486.448,E2 -15486.448} C_VEL
LIN {X 0,Y 312.784,Z 411.525,A -85,B 0,C 180,E1 -15489.049,E2 -15489.049} C_VEL
LIN {X 0,Y 312.631,Z 411.544,A -85,B 0,C 180,E1 -15492.991,E2 -15492.991} C_VEL
LIN {X 0,Y 312.634,Z 411.543,A -85,B 0,C 180,E1 -15495.65,E2 -15495.65} C_VEL
LIN {X 0,Y 312.627,Z 411.545,A -85,B 0,C 180,E1 -15499.237,E2 -15499.237} C_VEL
LIN {X 0,Y 312.542,Z 411.555,A -85,B 0,C 180,E1 -15502.79,E2 -15502.79} C_VEL
LIN {X 0,Y 312.6,Z 411.547,A -85,B 0,C 180,E1 -15505.936,E2 -15505.936} C_VEL
LIN {X 0,Y 312.542,Z 411.555,A -85,B 0,C 180,E1 -15509.65,E2 -15509.65} C_VEL
LIN {X 0,Y 312.517,Z 411.559,A -85,B 0,C 180,E1 -15513.69,E2 -15513.69} C_VEL
LIN {X 0,Y 312.55,Z 411.557,A -85,B 0,C 180,E1 -15517.382,E2 -15517.382} C_VEL
LIN {X 0,Y 312.533,Z 411.605,A -85,B 0,C 180,E1 -15519.024,E2 -15519.024} C_VEL
LIN {X 0,Y 313.035,Z 414.305,A -85,B 0,C 180,E1 -15522.341,E2 -15522.341} C_VEL
LIN {X 0,Y 313.569,Z 417.737,A -85,B 0,C 180,E1 -15525.99,E2 -15525.99} C_VEL
LIN {X 0,Y 314.168,Z 421.504,A -85,B 0,C 180,E1 -15529.555,E2 -15529.555} C_VEL
LIN {X 0,Y 314.526,Z 423.647,A -85,B 0,C 180,E1 -15531.45,E2 -15531.45} C_VEL
LIN {X 0,Y 314.63,Z 426.184,A -85,B 0,C 180,E1 -15533.528,E2 -15533.528} C_VEL
LIN {X 0,Y 314.111,Z 430.489,A -85,B 0,C 180,E1 -15536.759,E2 -15536.759} C_VEL
LIN {X 0,Y 313.083,Z 436.682,A -85,B 0,C 180,E1 -15541.1,E2 -15541.1} C_VEL
LIN {X 0,Y 312.379,Z 442.604,A -85,B 0,C 180,E1 -15545.049,E2 -15545.049} C_VEL
LIN {X 0,Y 312.354,Z 443.1,A -85,B 0,C 180,E1 -15545.266,E2 -15545.266} C_VEL
LIN {X 0,Y 313.976,Z 448.954,A -85,B 0,C 180,E1 -15545.679,E2 -15545.679} C_VEL
LIN {X 0,Y 316.827,Z 460.501,A -85,B 0,C 180,E1 -15546.607,E2 -15546.607} C_VEL
LIN {X 0,Y 318.899,Z 473.249,A -85,B 0,C 180,E1 -15547.761,E2 -15547.761} C_VEL
LIN {X 0,Y 319.75,Z 483.991,A -85,B 0,C 180,E1 -15548.878,E2 -15548.878} C_VEL
LIN {X 0,Y 319.626,Z 491.479,A -85,B 0,C 180,E1 -15549.739,E2 -15549.739} C_VEL
LIN {X 0,Y 317.817,Z 502.489,A -85,B 0,C 180,E1 -15551.132,E2 -15551.132} C_VEL
LIN {X 0,Y 316.279,Z 511.468,A -85,B 0,C 180,E1 -15552.544,E2 -15552.544} C_VEL
LIN {X 0,Y 314.943,Z 520.101,A -85,B 0,C 180,E1 -15554.212,E2 -15554.212} C_VEL
LIN {X 0,Y 313.544,Z 527.956,A -85,B 0,C 180,E1 -15556.058,E2 -15556.058} C_VEL
LIN {X 0,Y 312.52,Z 533.575,A -85,B 0,C 180,E1 -15557.665,E2 -15557.665} C_VEL
LIN {X 0,Y 311.715,Z 539.099,A -85,B 0,C 180,E1 -15559.609,E2 -15559.609} C_VEL
LIN {X 0,Y 311.153,Z 543.449,A -85,B 0,C 180,E1 -15561.558,E2 -15561.558} C_VEL
LIN {X 0,Y 310.831,Z 546.738,A -85,B 0,C 180,E1 -15563.509,E2 -15563.509} C_VEL
LIN {X 0,Y 310.717,Z 548.393,A -85,B 0,C 180,E1 -15564.81,E2 -15564.81} C_VEL
LIN {X 0,Y 310.722,Z 549.638,A -85,B 0,C 180,E1 -15566.11,E2 -15566.11} C_VEL
LIN {X 0,Y 310.702,Z 550.434,A -85,B 0,C 180,E1 -15567.408,E2 -15567.408} C_VEL
LIN {X 0,Y 310.711,Z 550.836,A -85,B 0,C 180,E1 -15568.704,E2 -15568.704} C_VEL
LIN {X 0,Y 310.763,Z 550.847,A -85,B 0,C 180,E1 -15570,E2 -15570} C_VEL
LIN {X 0,Y 310.719,Z 550.455,A -85,B 0,C 180,E1 -15571.297,E2 -15571.297} C_VEL
LIN {X 0,Y 310.716,Z 549.617,A -85,B 0,C 180,E1 -15572.593,E2 -15572.593} C_VEL
LIN {X 0,Y 310.746,Z 548.367,A -85,B 0,C 180,E1 -15573.891,E2 -15573.891} C_VEL
LIN {X 0,Y 310.767,Z 545.924,A -85,B 0,C 180,E1 -15575.694,E2 -15575.694} C_VEL
LIN {X 0,Y 311.01,Z 541.953,A -85,B 0,C 180,E1 -15577.793,E2 -15577.793} C_VEL
LIN {X 0,Y 311.427,Z 537.082,A -85,B 0,C 180,E1 -15579.745,E2 -15579.745} C_VEL
LIN {X 0,Y 312.042,Z 530.921,A -85,B 0,C 180,E1 -15581.696,E2 -15581.696} C_VEL
LIN {X 0,Y 313.101,Z 523.268,A -85,B 0,C 180,E1 -15583.633,E2 -15583.633} C_VEL
LIN {X 0,Y 314.115,Z 515.424,A -85,B 0,C 180,E1 -15585.242,E2 -15585.242} C_VEL
LIN {X 0,Y 315.195,Z 505.845,A -85,B 0,C 180,E1 -15586.85,E2 -15586.85} C_VEL
LIN {X 0,Y 316.511,Z 495.281,A -85,B 0,C 180,E1 -15588.279,E2 -15588.279} C_VEL
LIN {X 0,Y 317.515,Z 486.716,A -85,B 0,C 180,E1 -15589.224,E2 -15589.224} C_VEL
LIN {X 0,Y 316.509,Z 474.964,A -85,B 0,C 180,E1 -15590.381,E2 -15590.381} C_VEL
LIN {X 0,Y 314.838,Z 462.219,A -85,B 0,C 180,E1 -15591.385,E2 -15591.385} C_VEL
LIN {X 0,Y 312.481,Z 448.343,A -85,B 0,C 180,E1 -15592.215,E2 -15592.215} C_VEL
LIN {X 0,Y 311.814,Z 444.619,A -85,B 0,C 180,E1 -15592.398,E2 -15592.398} C_VEL
LIN {X 0,Y 312.271,Z 439.198,A -85,B 0,C 180,E1 -15595.809,E2 -15595.809} C_VEL
LIN {X 0,Y 313.018,Z 433.252,A -85,B 0,C 180,E1 -15599.601,E2 -15599.601} C_VEL
LIN {X 0,Y 313.737,Z 427.635,A -85,B 0,C 180,E1 -15603.287,E2 -15603.287} C_VEL
LIN {X 0,Y 314.144,Z 424.25,A -85,B 0,C 180,E1 -15605.568,E2 -15605.568} C_VEL
LIN {X 0,Y 314.017,Z 420.183,A -85,B 0,C 180,E1 -15608.433,E2 -15608.433} C_VEL
LIN {X 0,Y 313.401,Z 416.252,A -85,B 0,C 180,E1 -15611.371,E2 -15611.371} C_VEL
LIN {X 0,Y 312.477,Z 411.564,A -85,B 0,C 180,E1 -15615.173,E2 -15615.173} C_VEL
LIN {X 0,Y 312.486,Z 411.559,A -85,B 0,C 180,E1 -15617.919,E2 -15617.919} C_VEL
LIN {X 0,Y 312.5,Z 411.56,A -85,B 0,C 180,E1 -15620.971,E2 -15620.971} C_VEL
LIN {X 0,Y 312.533,Z 411.55,A -85,B 0,C 180,E1 -15624.22,E2 -15624.22} C_VEL
LIN {X 0,Y 312.506,Z 411.559,A -85,B 0,C 180,E1 -15627.334,E2 -15627.334} C_VEL
LIN {X 0,Y 312.553,Z 411.552,A -85,B 0,C 180,E1 -15631.276,E2 -15631.276} C_VEL
LIN {X 0,Y 312.587,Z 411.546,A -85,B 0,C 180,E1 -15634.711,E2 -15634.711} C_VEL
LIN {X 0,Y 312.589,Z 411.546,A -85,B 0,C 180,E1 -15637.529,E2 -15637.529} C_VEL
LIN {X 0,Y 312.639,Z 411.539,A -85,B 0,C 180,E1 -15641.656,E2 -15641.656} C_VEL
LIN {X 0,Y 312.695,Z 411.532,A -85,B 0,C 180,E1 -15645.686,E2 -15645.686} C_VEL
LIN {X 0,Y 312.703,Z 411.531,A -85,B 0,C 180,E1 -15649.642,E2 -15649.642} C_VEL
LIN {X 0,Y 312.873,Z 411.509,A -85,B 0,C 180,E1 -15652.254,E2 -15652.254} C_VEL
LIN {X 0,Y 312.718,Z 411.533,A -85,B 0,C 180,E1 -15654.842,E2 -15654.842} C_VEL
LIN {X 0,Y 312.989,Z 411.498,A -85,B 0,C 180,E1 -15658.713,E2 -15658.713} C_VEL
LIN {X 0,Y 312.991,Z 411.497,A -85,B 0,C 180,E1 -15661.287,E2 -15661.287} C_VEL
LIN {X 0,Y 312.718,Z 411.531,A -85,B 0,C 180,E1 -15665.158,E2 -15665.158} C_VEL
LIN {X 0,Y 312.873,Z 411.509,A -85,B 0,C 180,E1 -15667.746,E2 -15667.746} C_VEL
LIN {X 0,Y 312.67,Z 411.534,A -85,B 0,C 180,E1 -15671.671,E2 -15671.671} C_VEL
LIN {X 0,Y 312.701,Z 411.534,A -85,B 0,C 180,E1 -15674.887,E2 -15674.887} C_VEL
LIN {X 0,Y 312.632,Z 411.539,A -85,B 0,C 180,E1 -15679.237,E2 -15679.237} C_VEL
LIN {X 0,Y 312.547,Z 411.555,A -85,B 0,C 180,E1 -15682.789,E2 -15682.789} C_VEL
LIN {X 0,Y 312.584,Z 411.551,A -85,B 0,C 180,E1 -15686.723,E2 -15686.723} C_VEL
LIN {X 0,Y 312.546,Z 411.55,A -85,B 0,C 180,E1 -15689.65,E2 -15689.65} C_VEL
LIN {X 0,Y 312.52,Z 411.551,A -85,B 0,C 180,E1 -15693.689,E2 -15693.689} C_VEL
LIN {X 0,Y 312.526,Z 411.551,A -85,B 0,C 180,E1 -15697.385,E2 -15697.385} C_VEL
LIN {X 0,Y 312.491,Z 411.562,A -85,B 0,C 180,E1 -15700.709,E2 -15700.709} C_VEL
LIN {X 0,Y 312.452,Z 411.563,A -85,B 0,C 180,E1 -15704.21,E2 -15704.21} C_VEL
LIN {X 0,Y 312.485,Z 411.557,A -85,B 0,C 180,E1 -15707.919,E2 -15707.919} C_VEL
LIN {X 0,Y 312.537,Z 411.55,A -85,B 0,C 180,E1 -15711.91,E2 -15711.91} C_VEL
LIN {X 0,Y 312.508,Z 411.555,A -85,B 0,C 180,E1 -15715.79,E2 -15715.79} C_VEL
LIN {X 0,Y 312.522,Z 411.555,A -85,B 0,C 180,E1 -15718.853,E2 -15718.853} C_VEL
LIN {X 0,Y 312.572,Z 411.547,A -85,B 0,C 180,E1 -15721.824,E2 -15721.824} C_VEL
LIN {X 0,Y 312.587,Z 411.548,A -85,B 0,C 180,E1 -15724.711,E2 -15724.711} C_VEL
LIN {X 0,Y 312.589,Z 411.544,A -85,B 0,C 180,E1 -15727.529,E2 -15727.529} C_VEL
LIN {X 0,Y 312.64,Z 411.538,A -85,B 0,C 180,E1 -15731.656,E2 -15731.656} C_VEL
LIN {X 0,Y 312.696,Z 411.532,A -85,B 0,C 180,E1 -15735.686,E2 -15735.686} C_VEL
LIN {X 0,Y 312.704,Z 411.53,A -85,B 0,C 180,E1 -15739.642,E2 -15739.642} C_VEL
LIN {X 0,Y 312.876,Z 411.514,A -85,B 0,C 180,E1 -15742.254,E2 -15742.254} C_VEL
LIN {X 0,Y 312.718,Z 411.529,A -85,B 0,C 180,E1 -15744.842,E2 -15744.842} C_VEL
LIN {X 0,Y 312.99,Z 411.497,A -85,B 0,C 180,E1 -15748.713,E2 -15748.713} C_VEL
LIN {X 0,Y 312.99,Z 411.495,A -85,B 0,C 180,E1 -15751.286,E2 -15751.286} C_VEL
LIN {X 0,Y 312.688,Z 411.534,A -85,B 0,C 180,E1 -15753.866,E2 -15753.866} C_VEL
LIN {X 0,Y 312.737,Z 411.53,A -85,B 0,C 180,E1 -15756.451,E2 -15756.451} C_VEL
LIN {X 0,Y 312.321,Z 411.58,A -85,B 0,C 180,E1 -15759.062,E2 -15759.062} C_VEL
LIN {X 0,Y 312.085,Z 413.788,A -85,B 0,C 180,E1 -15761.693,E2 -15761.693} C_VEL
LIN {X 0,Y 311.935,Z 416.359,A -85,B 0,C 180,E1 -15764.349,E2 -15764.349} C_VEL
LIN {X 0,Y 311.51,Z 420.659,A -85,B 0,C 180,E1 -15768.636,E2 -15768.636} C_VEL
LIN {X 0,Y 311.39,Z 422.856,A -85,B 0,C 180,E1 -15770.692,E2 -15770.692} C_VEL
LIN {X 0,Y 314.741,Z 436.282,A -85,B 0,C 180,E1 -15771.532,E2 -15771.532} C_VEL
LIN {X 0,Y 317.198,Z 448.035,A -85,B 0,C 180,E1 -15772.469,E2 -15772.469} C_VEL
LIN {X 0,Y 318.762,Z 457.587,A -85,B 0,C 180,E1 -15773.381,E2 -15773.381} C_VEL
LIN {X 0,Y 317.608,Z 468.708,A -85,B 0,C 180,E1 -15774.512,E2 -15774.512} C_VEL
LIN {X 0,Y 316.443,Z 479.117,A -85,B 0,C 180,E1 -15775.839,E2 -15775.839} C_VEL
LIN {X 0,Y 315.129,Z 489.137,A -85,B 0,C 180,E1 -15777.43,E2 -15777.43} C_VEL
LIN {X 0,Y 314.025,Z 498.18,A -85,B 0,C 180,E1 -15779.21,E2 -15779.21} C_VEL
LIN {X 0,Y 312.961,Z 505.944,A -85,B 0,C 180,E1 -15781.097,E2 -15781.097} C_VEL
LIN {X 0,Y 312.13,Z 512.519,A -85,B 0,C 180,E1 -15783.114,E2 -15783.114} C_VEL
LIN {X 0,Y 311.54,Z 517.352,A -85,B 0,C 180,E1 -15784.977,E2 -15784.977} C_VEL
LIN {X 0,Y 311.118,Z 521.018,A -85,B 0,C 180,E1 -15786.77,E2 -15786.77} C_VEL
LIN {X 0,Y 310.841,Z 523.628,A -85,B 0,C 180,E1 -15788.454,E2 -15788.454} C_VEL
LIN {X 0,Y 310.646,Z 525.124,A -85,B 0,C 180,E1 -15789.717,E2 -15789.717} C_VEL
LIN {X 0,Y 310.546,Z 526.645,A -85,B 0,C 180,E1 -15791.684,E2 -15791.684} C_VEL
LIN {X 0,Y 310.505,Z 527.224,A -85,B 0,C 180,E1 -15793.59,E2 -15793.59} C_VEL
LIN {X 0,Y 310.579,Z 526.963,A -85,B 0,C 180,E1 -15795.453,E2 -15795.453} C_VEL
LIN {X 0,Y 310.813,Z 525.915,A -85,B 0,C 180,E1 -15797.285,E2 -15797.285} C_VEL
LIN {X 0,Y 311.194,Z 524.108,A -85,B 0,C 180,E1 -15799.085,E2 -15799.085} C_VEL
LIN {X 0,Y 311.885,Z 520.369,A -85,B 0,C 180,E1 -15801.487,E2 -15801.487} C_VEL
LIN {X 0,Y 312.913,Z 514.882,A -85,B 0,C 180,E1 -15803.954,E2 -15803.954} C_VEL
LIN {X 0,Y 313.994,Z 508.882,A -85,B 0,C 180,E1 -15805.974,E2 -15805.974} C_VEL
LIN {X 0,Y 315.353,Z 501.804,A -85,B 0,C 180,E1 -15807.872,E2 -15807.872} C_VEL
LIN {X 0,Y 316.891,Z 493.733,A -85,B 0,C 180,E1 -15809.617,E2 -15809.617} C_VEL
LIN {X 0,Y 318.449,Z 484.796,A -85,B 0,C 180,E1 -15811.194,E2 -15811.194} C_VEL
LIN {X 0,Y 319.925,Z 475.524,A -85,B 0,C 180,E1 -15812.528,E2 -15812.528} C_VEL
LIN {X 0,Y 321.347,Z 465.285,A -85,B 0,C 180,E1 -15813.724,E2 -15813.724} C_VEL
LIN {X 0,Y 321.782,Z 460.329,A -85,B 0,C 180,E1 -15814.234,E2 -15814.234} C_VEL
LIN {X 0,Y 319.733,Z 449.136,A -85,B 0,C 180,E1 -15815.467,E2 -15815.467} C_VEL
LIN {X 0,Y 316.685,Z 437.962,A -85,B 0,C 180,E1 -15816.585,E2 -15816.585} C_VEL
LIN {X 0,Y 316.041,Z 435.92,A -85,B 0,C 180,E1 -15816.781,E2 -15816.781} C_VEL
LIN {X 0,Y 314.669,Z 432.935,A -85,B 0,C 180,E1 -15817.143,E2 -15817.143} C_VEL
LIN {X 0,Y 312.136,Z 429.341,A -85,B 0,C 180,E1 -15817.832,E2 -15817.832} C_VEL
LIN {X 0,Y 308.678,Z 425.921,A -85,B 0,C 180,E1 -15818.956,E2 -15818.956} C_VEL
LIN {X 0,Y 306.052,Z 423.665,A -85,B 0,C 180,E1 -15820.268,E2 -15820.268} C_VEL
LIN {X 0,Y 305.329,Z 422.553,A -85,B 0,C 180,E1 -15821.337,E2 -15821.337} C_VEL
LIN {X 0,Y 305.791,Z 419.29,A -85,B 0,C 180,E1 -15825.356,E2 -15825.356} C_VEL
LIN {X 0,Y 306.059,Z 416.247,A -85,B 0,C 180,E1 -15829.415,E2 -15829.415} C_VEL
LIN {X 0,Y 306.126,Z 414.405,A -85,B 0,C 180,E1 -15832.083,E2 -15832.083} C_VEL
LIN {X 0,Y 305.738,Z 412.783,A -85,B 0,C 180,E1 -15834.724,E2 -15834.724} C_VEL
LIN {X 0,Y 305.883,Z 412.385,A -85,B 0,C 180,E1 -15837.366,E2 -15837.366} C_VEL
LIN {X 0,Y 306.07,Z 412.361,A -85,B 0,C 180,E1 -15840,E2 -15840} C_VEL
LIN {X 0,Y 305.883,Z 412.382,A -85,B 0,C 180,E1 -15842.634,E2 -15842.634} C_VEL
LIN {X 0,Y 305.848,Z 412.389,A -85,B 0,C 180,E1 -15846.598,E2 -15846.598} C_VEL
LIN {X 0,Y 305.732,Z 412.403,A -85,B 0,C 180,E1 -15849.26,E2 -15849.26} C_VEL
LIN {X 0,Y 305.585,Z 412.421,A -85,B 0,C 180,E1 -15853.296,E2 -15853.296} C_VEL
LIN {X 0,Y 305.59,Z 412.42,A -85,B 0,C 180,E1 -15856.02,E2 -15856.02} C_VEL
LIN {X 0,Y 305.573,Z 412.423,A -85,B 0,C 180,E1 -15859.445,E2 -15859.445} C_VEL
LIN {X 0,Y 305.487,Z 412.434,A -85,B 0,C 180,E1 -15863.042,E2 -15863.042} C_VEL
LIN {X 0,Y 305.545,Z 412.426,A -85,B 0,C 180,E1 -15866.228,E2 -15866.228} C_VEL
LIN {X 0,Y 305.493,Z 412.433,A -85,B 0,C 180,E1 -15869.051,E2 -15869.051} C_VEL
LIN {X 0,Y 305.442,Z 412.441,A -85,B 0,C 180,E1 -15871.953,E2 -15871.953} C_VEL
LIN {X 0,Y 305.46,Z 412.44,A -85,B 0,C 180,E1 -15875.114,E2 -15875.114} C_VEL
LIN {X 0,Y 305.535,Z 412.735,A -85,B 0,C 180,E1 -15878.394,E2 -15878.394} C_VEL
LIN {X 0,Y 306,Z 415.343,A -85,B 0,C 180,E1 -15881.763,E2 -15881.763} C_VEL
LIN {X 0,Y 306.503,Z 418.508,A -85,B 0,C 180,E1 -15885.302,E2 -15885.302} C_VEL
LIN {X 0,Y 307.113,Z 422.285,A -85,B 0,C 180,E1 -15889.041,E2 -15889.041} C_VEL
LIN {X 0,Y 307.568,Z 425.46,A -85,B 0,C 180,E1 -15891.907,E2 -15891.907} C_VEL
LIN {X 0,Y 307.559,Z 428.459,A -85,B 0,C 180,E1 -15894.36,E2 -15894.36} C_VEL
LIN {X 0,Y 306.795,Z 433.23,A -85,B 0,C 180,E1 -15897.951,E2 -15897.951} C_VEL
LIN {X 0,Y 305.757,Z 439.864,A -85,B 0,C 180,E1 -15902.632,E2 -15902.632} C_VEL
LIN {X 0,Y 305.403,Z 442.591,A -85,B 0,C 180,E1 -15904.497,E2 -15904.497} C_VEL
LIN {X 0,Y 308.03,Z 451.883,A -85,B 0,C 180,E1 -15905.219,E2 -15905.219} C_VEL
LIN {X 0,Y 310.771,Z 463.878,A -85,B 0,C 180,E1 -15906.262,E2 -15906.262} C_VEL
LIN {X 0,Y 312.582,Z 476.732,A -85,B 0,C 180,E1 -15907.529,E2 -15907.529} C_VEL
LIN {X 0,Y 313.144,Z 487.034,A -85,B 0,C 180,E1 -15908.687,E2 -15908.687} C_VEL
LIN {X 0,Y 312.828,Z 493.309,A -85,B 0,C 180,E1 -15909.45,E2 -15909.45} C_VEL
LIN {X 0,Y 310.733,Z 504.934,A -85,B 0,C 180,E1 -15911.027,E2 -15911.027} C_VEL
LIN {X 0,Y 309.18,Z 513.472,A -85,B 0,C 180,E1 -15912.472,E2 -15912.472} C_VEL
LIN {X 0,Y 307.877,Z 521.397,A -85,B 0,C 180,E1 -15914.103,E2 -15914.103} C_VEL
LIN {X 0,Y 306.445,Z 529.218,A -85,B 0,C 180,E1 -15916.066,E2 -15916.066} C_VEL
LIN {X 0,Y 305.21,Z 535.523,A -85,B 0,C 180,E1 -15918.04,E2 -15918.04} C_VEL
LIN {X 0,Y 304.465,Z 540.578,A -85,B 0,C 180,E1 -15920.031,E2 -15920.031} C_VEL
LIN {X 0,Y 303.957,Z 544.522,A -85,B 0,C 180,E1 -15922.026,E2 -15922.026} C_VEL
LIN {X 0,Y 303.66,Z 547.864,A -85,B 0,C 180,E1 -15924.389,E2 -15924.389} C_VEL
LIN {X 0,Y 303.635,Z 549.415,A -85,B 0,C 180,E1 -15926.019,E2 -15926.019} C_VEL
LIN {X 0,Y 303.625,Z 550.188,A -85,B 0,C 180,E1 -15927.347,E2 -15927.347} C_VEL
LIN {X 0,Y 303.624,Z 550.57,A -85,B 0,C 180,E1 -15928.674,E2 -15928.674} C_VEL
LIN {X 0,Y 303.672,Z 550.562,A -85,B 0,C 180,E1 -15930.001,E2 -15930.001} C_VEL
LIN {X 0,Y 303.632,Z 550.134,A -85,B 0,C 180,E1 -15931.327,E2 -15931.327} C_VEL
LIN {X 0,Y 303.64,Z 549.269,A -85,B 0,C 180,E1 -15932.654,E2 -15932.654} C_VEL
LIN {X 0,Y 303.657,Z 547.998,A -85,B 0,C 180,E1 -15933.982,E2 -15933.982} C_VEL
LIN {X 0,Y 303.662,Z 545.853,A -85,B 0,C 180,E1 -15935.614,E2 -15935.614} C_VEL
LIN {X 0,Y 303.948,Z 541.493,A -85,B 0,C 180,E1 -15937.975,E2 -15937.975} C_VEL
LIN {X 0,Y 304.395,Z 536.57,A -85,B 0,C 180,E1 -15939.972,E2 -15939.972} C_VEL
LIN {X 0,Y 305.05,Z 530.353,A -85,B 0,C 180,E1 -15941.967,E2 -15941.967} C_VEL
LIN {X 0,Y 306.156,Z 522.61,A -85,B 0,C 180,E1 -15943.948,E2 -15943.948} C_VEL
LIN {X 0,Y 307.414,Z 512.885,A -85,B 0,C 180,E1 -15945.923,E2 -15945.923} C_VEL
LIN {X 0,Y 308.639,Z 502.854,A -85,B 0,C 180,E1 -15947.561,E2 -15947.561} C_VEL
LIN {X 0,Y 310.117,Z 491.572,A -85,B 0,C 180,E1 -15949.013,E2 -15949.013} C_VEL
LIN {X 0,Y 310.567,Z 487.164,A -85,B 0,C 180,E1 -15949.499,E2 -15949.499} C_VEL
LIN {X 0,Y 309.569,Z 475.399,A -85,B 0,C 180,E1 -15950.7,E2 -15950.7} C_VEL
LIN {X 0,Y 307.974,Z 463.096,A -85,B 0,C 180,E1 -15951.718,E2 -15951.718} C_VEL
LIN {X 0,Y 305.792,Z 449.877,A -85,B 0,C 180,E1 -15952.557,E2 -15952.557} C_VEL
LIN {X 0,Y 304.775,Z 444.388,A -85,B 0,C 180,E1 -15952.847,E2 -15952.847} C_VEL
LIN {X 0,Y 305.235,Z 439.32,A -85,B 0,C 180,E1 -15956.107,E2 -15956.107} C_VEL
LIN {X 0,Y 305.868,Z 434.619,A -85,B 0,C 180,E1 -15959.175,E2 -15959.175} C_VEL
LIN {X 0,Y 306.714,Z 428.38,A -85,B 0,C 180,E1 -15963.363,E2 -15963.363} C_VEL
LIN {X 0,Y 307.11,Z 424.982,A -85,B 0,C 180,E1 -15965.701,E2 -15965.701} C_VEL
LIN {X 0,Y 306.957,Z 420.605,A -85,B 0,C 180,E1 -15968.88,E2 -15968.88} C_VEL
LIN {X 0,Y 306.05,Z 415.668,A -85,B 0,C 180,E1 -15972.706,E2 -15972.706} C_VEL
LIN {X 0,Y 305.424,Z 412.442,A -85,B 0,C 180,E1 -15975.507,E2 -15975.507} C_VEL
LIN {X 0,Y 305.456,Z 412.438,A -85,B 0,C 180,E1 -15979.4,E2 -15979.4} C_VEL
LIN {X 0,Y 305.474,Z 412.435,A -85,B 0,C 180,E1 -15983.26,E2 -15983.26} C_VEL
LIN {X 0,Y 305.466,Z 412.432,A -85,B 0,C 180,E1 -15986.483,E2 -15986.483} C_VEL
LIN {X 0,Y 305.497,Z 412.431,A -85,B 0,C 180,E1 -15990.95,E2 -15990.95} C_VEL
LIN {X 0,Y 305.567,Z 412.418,A -85,B 0,C 180,E1 -15994.087,E2 -15994.087} C_VEL
LIN {X 0,Y 305.501,Z 412.428,A -85,B 0,C 180,E1 -15998.403,E2 -15998.403} C_VEL
LIN {X 0,Y 305.591,Z 412.42,A -85,B 0,C 180,E1 -16001.218,E2 -16001.218} C_VEL
LIN {X 0,Y 305.65,Z 412.412,A -85,B 0,C 180,E1 -16005.349,E2 -16005.349} C_VEL
LIN {X 0,Y 305.64,Z 412.412,A -85,B 0,C 180,E1 -16009.4,E2 -16009.4} C_VEL
LIN {X 0,Y 305.814,Z 412.388,A -85,B 0,C 180,E1 -16012.074,E2 -16012.074} C_VEL
LIN {X 0,Y 305.689,Z 412.407,A -85,B 0,C 180,E1 -16014.723,E2 -16014.723} C_VEL
LIN {X 0,Y 305.956,Z 412.373,A -85,B 0,C 180,E1 -16018.684,E2 -16018.684} C_VEL
LIN {X 0,Y 305.958,Z 412.372,A -85,B 0,C 180,E1 -16021.316,E2 -16021.316} C_VEL
LIN {X 0,Y 305.852,Z 412.386,A -85,B 0,C 180,E1 -16026.608,E2 -16026.608} C_VEL
LIN {X 0,Y 305.737,Z 412.4,A -85,B 0,C 180,E1 -16029.26,E2 -16029.26} C_VEL
LIN {X 0,Y 305.59,Z 412.417,A -85,B 0,C 180,E1 -16033.296,E2 -16033.296} C_VEL
LIN {X 0,Y 305.595,Z 412.413,A -85,B 0,C 180,E1 -16036.02,E2 -16036.02} C_VEL
LIN {X 0,Y 305.578,Z 412.416,A -85,B 0,C 180,E1 -16039.445,E2 -16039.445} C_VEL
LIN {X 0,Y 305.491,Z 412.431,A -85,B 0,C 180,E1 -16043.041,E2 -16043.041} C_VEL
LIN {X 0,Y 305.555,Z 412.422,A -85,B 0,C 180,E1 -16046.229,E2 -16046.229} C_VEL
LIN {X 0,Y 305.497,Z 412.43,A -85,B 0,C 180,E1 -16049.05,E2 -16049.05} C_VEL
LIN {X 0,Y 305.466,Z 412.43,A -85,B 0,C 180,E1 -16053.517,E2 -16053.517} C_VEL
LIN {X 0,Y 305.476,Z 412.433,A -85,B 0,C 180,E1 -16056.739,E2 -16056.739} C_VEL
LIN {X 0,Y 305.455,Z 412.437,A -85,B 0,C 180,E1 -16060.6,E2 -16060.6} C_VEL
LIN {X 0,Y 305.426,Z 412.437,A -85,B 0,C 180,E1 -16063.655,E2 -16063.655} C_VEL
LIN {X 0,Y 305.456,Z 412.432,A -85,B 0,C 180,E1 -16067.414,E2 -16067.414} C_VEL
LIN {X 0,Y 305.497,Z 412.426,A -85,B 0,C 180,E1 -16071.6,E2 -16071.6} C_VEL
LIN {X 0,Y 305.464,Z 412.434,A -85,B 0,C 180,E1 -16074.887,E2 -16074.887} C_VEL
LIN {X 0,Y 305.451,Z 412.438,A -85,B 0,C 180,E1 -16078.355,E2 -16078.355} C_VEL
LIN {X 0,Y 305.514,Z 412.426,A -85,B 0,C 180,E1 -16081.113,E2 -16081.113} C_VEL
LIN {X 0,Y 305.567,Z 412.42,A -85,B 0,C 180,E1 -16084.087,E2 -16084.087} C_VEL
LIN {X 0,Y 305.528,Z 412.429,A -85,B 0,C 180,E1 -16088.405,E2 -16088.405} C_VEL
LIN {X 0,Y 305.592,Z 412.415,A -85,B 0,C 180,E1 -16091.217,E2 -16091.217} C_VEL
LIN {X 0,Y 305.651,Z 412.409,A -85,B 0,C 180,E1 -16095.349,E2 -16095.349} C_VEL
LIN {X 0,Y 305.64,Z 412.41,A -85,B 0,C 180,E1 -16099.399,E2 -16099.399} C_VEL
LIN {X 0,Y 305.817,Z 412.391,A -85,B 0,C 180,E1 -16102.074,E2 -16102.074} C_VEL
LIN {X 0,Y 305.69,Z 412.405,A -85,B 0,C 180,E1 -16104.723,E2 -16104.723} C_VEL
LIN {X 0,Y 305.957,Z 412.373,A -85,B 0,C 180,E1 -16108.683,E2 -16108.683} C_VEL
LIN {X 0,Y 305.957,Z 412.371,A -85,B 0,C 180,E1 -16111.316,E2 -16111.316} C_VEL
LIN {X 0,Y 305.646,Z 412.41,A -85,B 0,C 180,E1 -16115.277,E2 -16115.277} C_VEL
LIN {X 0,Y 305.497,Z 412.431,A -85,B 0,C 180,E1 -16117.933,E2 -16117.933} C_VEL
LIN {X 0,Y 305.231,Z 412.464,A -85,B 0,C 180,E1 -16119.275,E2 -16119.275} C_VEL
LIN {X 0,Y 304.948,Z 416.215,A -85,B 0,C 180,E1 -16123.324,E2 -16123.324} C_VEL
LIN {X 0,Y 304.658,Z 418.897,A -85,B 0,C 180,E1 -16126.07,E2 -16126.07} C_VEL
LIN {X 0,Y 304.348,Z 423.023,A -85,B 0,C 180,E1 -16130.221,E2 -16130.221} C_VEL
LIN {X 0,Y 308.084,Z 438.127,A -85,B 0,C 180,E1 -16131.231,E2 -16131.231} C_VEL
LIN {X 0,Y 310.585,Z 450.455,A -85,B 0,C 180,E1 -16132.272,E2 -16132.272} C_VEL
LIN {X 0,Y 311.856,Z 458.163,A -85,B 0,C 180,E1 -16133.051,E2 -16133.051} C_VEL
LIN {X 0,Y 310.629,Z 470.298,A -85,B 0,C 180,E1 -16134.335,E2 -16134.335} C_VEL
LIN {X 0,Y 309.345,Z 480.823,A -85,B 0,C 180,E1 -16135.753,E2 -16135.753} C_VEL
LIN {X 0,Y 307.957,Z 491.378,A -85,B 0,C 180,E1 -16137.523,E2 -16137.523} C_VEL
LIN {X 0,Y 306.745,Z 500.558,A -85,B 0,C 180,E1 -16139.467,E2 -16139.467} C_VEL
LIN {X 0,Y 305.726,Z 507.718,A -85,B 0,C 180,E1 -16141.348,E2 -16141.348} C_VEL
LIN {X 0,Y 304.873,Z 514.499,A -85,B 0,C 180,E1 -16143.59,E2 -16143.59} C_VEL
LIN {X 0,Y 304.203,Z 520.038,A -85,B 0,C 180,E1 -16146.04,E2 -16146.04} C_VEL
LIN {X 0,Y 303.717,Z 524.211,A -85,B 0,C 180,E1 -16148.665,E2 -16148.665} C_VEL
LIN {X 0,Y 303.495,Z 526.01,A -85,B 0,C 180,E1 -16150.42,E2 -16150.42} C_VEL
LIN {X 0,Y 303.427,Z 527.116,A -85,B 0,C 180,E1 -16152.197,E2 -16152.197} C_VEL
LIN {X 0,Y 303.42,Z 527.521,A -85,B 0,C 180,E1 -16154.107,E2 -16154.107} C_VEL
LIN {X 0,Y 303.541,Z 527.106,A -85,B 0,C 180,E1 -16156.005,E2 -16156.005} C_VEL
LIN {X 0,Y 303.843,Z 525.866,A -85,B 0,C 180,E1 -16157.873,E2 -16157.873} C_VEL
LIN {X 0,Y 304.561,Z 522.589,A -85,B 0,C 180,E1 -16160.611,E2 -16160.611} C_VEL
LIN {X 0,Y 305.153,Z 519.389,A -85,B 0,C 180,E1 -16162.437,E2 -16162.437} C_VEL
LIN {X 0,Y 306.004,Z 515.168,A -85,B 0,C 180,E1 -16164.297,E2 -16164.297} C_VEL
LIN {X 0,Y 307.051,Z 509.861,A -85,B 0,C 180,E1 -16166.156,E2 -16166.156} C_VEL
LIN {X 0,Y 308.367,Z 503.313,A -85,B 0,C 180,E1 -16168.002,E2 -16168.002} C_VEL
LIN {X 0,Y 309.975,Z 495.209,A -85,B 0,C 180,E1 -16169.843,E2 -16169.843} C_VEL
LIN {X 0,Y 311.72,Z 485.889,A -85,B 0,C 180,E1 -16171.555,E2 -16171.555} C_VEL
LIN {X 0,Y 313.344,Z 476.269,A -85,B 0,C 180,E1 -16172.987,E2 -16172.987} C_VEL
LIN {X 0,Y 314.942,Z 465.489,A -85,B 0,C 180,E1 -16174.274,E2 -16174.274} C_VEL
LIN {X 0,Y 315.281,Z 462.232,A -85,B 0,C 180,E1 -16174.623,E2 -16174.623} C_VEL
LIN {X 0,Y 313.301,Z 450.895,A -85,B 0,C 180,E1 -16175.951,E2 -16175.951} C_VEL
LIN {X 0,Y 310.178,Z 439.318,A -85,B 0,C 180,E1 -16177.169,E2 -16177.169} C_VEL
LIN {X 0,Y 305.727,Z 427.33,A -85,B 0,C 180,E1 -16178.339,E2 -16178.339} C_VEL
LIN {X 0,Y 305.07,Z 424.928,A -85,B 0,C 180,E1 -16178.548,E2 -16178.548} C_VEL
LIN {X 0,Y 305.329,Z 422.553,A -85,B 0,C 180,E1 -16181.337,E2 -16181.337} C_VEL
LIN {X 0,Y 304.729,Z 421.762,A -85,B 0,C 180,E1 -16182.431,E2 -16182.431} C_VEL
LIN {X 0,Y 302.071,Z 420.777,A -85,B 0,C 180,E1 -16184.227,E2 -16184.227} C_VEL
LIN {X 0,Y 299.84,Z 420.039,A -85,B 0,C 180,E1 -16185.684,E2 -16185.684} C_VEL
LIN {X 0,Y 298.936,Z 419.364,A -85,B 0,C 180,E1 -16186.805,E2 -16186.805} C_VEL
LIN {X 0,Y 298.89,Z 419.097,A -85,B 0,C 180,E1 -16187.183,E2 -16187.183} C_VEL
LIN {X 0,Y 299.128,Z 416.637,A -85,B 0,C 180,E1 -16190.67,E2 -16190.67} C_VEL
LIN {X 0,Y 299.054,Z 414.97,A -85,B 0,C 180,E1 -16193.252,E2 -16193.252} C_VEL
LIN {X 0,Y 298.619,Z 413.45,A -85,B 0,C 180,E1 -16195.951,E2 -16195.951} C_VEL
LIN {X 0,Y 298.922,Z 413.252,A -85,B 0,C 180,E1 -16198.653,E2 -16198.653} C_VEL
LIN {X 0,Y 298.922,Z 413.253,A -85,B 0,C 180,E1 -16201.347,E2 -16201.347} C_VEL
LIN {X 0,Y 298.794,Z 413.268,A -85,B 0,C 180,E1 -16206.754,E2 -16206.754} C_VEL
LIN {X 0,Y 298.677,Z 413.281,A -85,B 0,C 180,E1 -16209.481,E2 -16209.481} C_VEL
LIN {X 0,Y 298.548,Z 413.298,A -85,B 0,C 180,E1 -16213.616,E2 -16213.616} C_VEL
LIN {X 0,Y 298.545,Z 413.299,A -85,B 0,C 180,E1 -16216.409,E2 -16216.409} C_VEL
LIN {X 0,Y 298.508,Z 413.302,A -85,B 0,C 180,E1 -16219.655,E2 -16219.655} C_VEL
LIN {X 0,Y 298.454,Z 413.307,A -85,B 0,C 180,E1 -16223.598,E2 -16223.598} C_VEL
LIN {X 0,Y 298.486,Z 413.307,A -85,B 0,C 180,E1 -16226.575,E2 -16226.575} C_VEL
LIN {X 0,Y 298.418,Z 413.314,A -85,B 0,C 180,E1 -16229.641,E2 -16229.641} C_VEL
LIN {X 0,Y 298.393,Z 413.318,A -85,B 0,C 180,E1 -16232.801,E2 -16232.801} C_VEL
LIN {X 0,Y 298.468,Z 413.311,A -85,B 0,C 180,E1 -16236.815,E2 -16236.815} C_VEL
LIN {X 0,Y 298.99,Z 416.403,A -85,B 0,C 180,E1 -16241.16,E2 -16241.16} C_VEL
LIN {X 0,Y 299.564,Z 419.932,A -85,B 0,C 180,E1 -16245.267,E2 -16245.267} C_VEL
LIN {X 0,Y 300.163,Z 423.623,A -85,B 0,C 180,E1 -16249.037,E2 -16249.037} C_VEL
LIN {X 0,Y 300.445,Z 425.548,A -85,B 0,C 180,E1 -16250.834,E2 -16250.834} C_VEL
LIN {X 0,Y 300.615,Z 427.585,A -85,B 0,C 180,E1 -16252.644,E2 -16252.644} C_VEL
LIN {X 0,Y 300.447,Z 430.407,A -85,B 0,C 180,E1 -16254.957,E2 -16254.957} C_VEL
LIN {X 0,Y 299.858,Z 433.758,A -85,B 0,C 180,E1 -16257.54,E2 -16257.54} C_VEL
LIN {X 0,Y 298.808,Z 439.787,A -85,B 0,C 180,E1 -16261.94,E2 -16261.94} C_VEL
LIN {X 0,Y 298.528,Z 442.437,A -85,B 0,C 180,E1 -16263.707,E2 -16263.707} C_VEL
LIN {X 0,Y 301.306,Z 451.997,A -85,B 0,C 180,E1 -16264.498,E2 -16264.498} C_VEL
LIN {X 0,Y 303.997,Z 463.369,A -85,B 0,C 180,E1 -16265.547,E2 -16265.547} C_VEL
LIN {X 0,Y 305.818,Z 475.848,A -85,B 0,C 180,E1 -16266.816,E2 -16266.816} C_VEL
LIN {X 0,Y 306.527,Z 486.656,A -85,B 0,C 180,E1 -16268.072,E2 -16268.072} C_VEL
LIN {X 0,Y 306.205,Z 493.827,A -85,B 0,C 180,E1 -16268.985,E2 -16268.985} C_VEL
LIN {X 0,Y 304.216,Z 504.223,A -85,B 0,C 180,E1 -16270.429,E2 -16270.429} C_VEL
LIN {X 0,Y 302.421,Z 513.7,A -85,B 0,C 180,E1 -16272.067,E2 -16272.067} C_VEL
LIN {X 0,Y 300.765,Z 522.919,A -85,B 0,C 180,E1 -16274.065,E2 -16274.065} C_VEL
LIN {X 0,Y 299.319,Z 530.388,A -85,B 0,C 180,E1 -16276.075,E2 -16276.075} C_VEL
LIN {X 0,Y 298.234,Z 535.506,A -85,B 0,C 180,E1 -16277.756,E2 -16277.756} C_VEL
LIN {X 0,Y 297.445,Z 540.503,A -85,B 0,C 180,E1 -16279.793,E2 -16279.793} C_VEL
LIN {X 0,Y 296.898,Z 544.388,A -85,B 0,C 180,E1 -16281.835,E2 -16281.835} C_VEL
LIN {X 0,Y 296.581,Z 547.868,A -85,B 0,C 180,E1 -16284.424,E2 -16284.424} C_VEL
LIN {X 0,Y 296.532,Z 549.188,A -85,B 0,C 180,E1 -16285.923,E2 -16285.923} C_VEL
LIN {X 0,Y 296.55,Z 549.943,A -85,B 0,C 180,E1 -16287.284,E2 -16287.284} C_VEL
LIN {X 0,Y 296.54,Z 550.305,A -85,B 0,C 180,E1 -16288.642,E2 -16288.642} C_VEL
LIN {X 0,Y 296.584,Z 550.276,A -85,B 0,C 180,E1 -16290.001,E2 -16290.001} C_VEL
LIN {X 0,Y 296.548,Z 549.808,A -85,B 0,C 180,E1 -16291.359,E2 -16291.359} C_VEL
LIN {X 0,Y 296.564,Z 548.921,A -85,B 0,C 180,E1 -16292.717,E2 -16292.717} C_VEL
LIN {X 0,Y 296.57,Z 547.628,A -85,B 0,C 180,E1 -16294.077,E2 -16294.077} C_VEL
LIN {X 0,Y 296.589,Z 545.683,A -85,B 0,C 180,E1 -16295.593,E2 -16295.593} C_VEL
LIN {X 0,Y 296.888,Z 541.027,A -85,B 0,C 180,E1 -16298.166,E2 -16298.166} C_VEL
LIN {X 0,Y 297.38,Z 536.052,A -85,B 0,C 180,E1 -16300.21,E2 -16300.21} C_VEL
LIN {X 0,Y 298.06,Z 529.774,A -85,B 0,C 180,E1 -16302.252,E2 -16302.252} C_VEL
LIN {X 0,Y 299.188,Z 521.927,A -85,B 0,C 180,E1 -16304.28,E2 -16304.28} C_VEL
LIN {X 0,Y 300.308,Z 513.914,A -85,B 0,C 180,E1 -16305.961,E2 -16305.961} C_VEL
LIN {X 0,Y 301.556,Z 504.148,A -85,B 0,C 180,E1 -16307.637,E2 -16307.637} C_VEL
LIN {X 0,Y 302.995,Z 493.341,A -85,B 0,C 180,E1 -16309.125,E2 -16309.125} C_VEL
LIN {X 0,Y 303.6,Z 487.593,A -85,B 0,C 180,E1 -16309.789,E2 -16309.789} C_VEL
LIN {X 0,Y 302.566,Z 475.029,A -85,B 0,C 180,E1 -16311.11,E2 -16311.11} C_VEL
LIN {X 0,Y 300.934,Z 462.419,A -85,B 0,C 180,E1 -16312.178,E2 -16312.178} C_VEL
LIN {X 0,Y 298.56,Z 448.568,A -85,B 0,C 180,E1 -16313.073,E2 -16313.073} C_VEL
LIN {X 0,Y 297.768,Z 444.065,A -85,B 0,C 180,E1 -16313.346,E2 -16313.346} C_VEL
LIN {X 0,Y 298.568,Z 436.949,A -85,B 0,C 180,E1 -16318.085,E2 -16318.085} C_VEL
LIN {X 0,Y 299.172,Z 432.462,A -85,B 0,C 180,E1 -16321.119,E2 -16321.119} C_VEL
LIN {X 0,Y 299.974,Z 427.014,A -85,B 0,C 180,E1 -16324.914,E2 -16324.914} C_VEL
LIN {X 0,Y 300.023,Z 423.431,A -85,B 0,C 180,E1 -16327.521,E2 -16327.521} C_VEL
LIN {X 0,Y 299.649,Z 419.976,A -85,B 0,C 180,E1 -16330.164,E2 -16330.164} C_VEL
LIN {X 0,Y 298.701,Z 415.056,A -85,B 0,C 180,E1 -16334.142,E2 -16334.142} C_VEL
LIN {X 0,Y 298.388,Z 413.319,A -85,B 0,C 180,E1 -16335.753,E2 -16335.753} C_VEL
LIN {X 0,Y 298.389,Z 413.318,A -85,B 0,C 180,E1 -16338.912,E2 -16338.912} C_VEL
LIN {X 0,Y 298.446,Z 413.31,A -85,B 0,C 180,E1 -16343.193,E2 -16343.193} C_VEL
LIN {X 0,Y 298.397,Z 413.318,A -85,B 0,C 180,E1 -16347.2,E2 -16347.2} C_VEL
LIN {X 0,Y 298.433,Z 413.309,A -85,B 0,C 180,E1 -16350.615,E2 -16350.615} C_VEL
LIN {X 0,Y 298.479,Z 413.303,A -85,B 0,C 180,E1 -16353.477,E2 -16353.477} C_VEL
LIN {X 0,Y 298.436,Z 413.309,A -85,B 0,C 180,E1 -16356.697,E2 -16356.697} C_VEL
LIN {X 0,Y 298.54,Z 413.297,A -85,B 0,C 180,E1 -16360.757,E2 -16360.757} C_VEL
LIN {X 0,Y 298.595,Z 413.293,A -85,B 0,C 180,E1 -16364.995,E2 -16364.995} C_VEL
LIN {X 0,Y 298.595,Z 413.291,A -85,B 0,C 180,E1 -16369.147,E2 -16369.147} C_VEL
LIN {X 0,Y 298.76,Z 413.267,A -85,B 0,C 180,E1 -16371.886,E2 -16371.886} C_VEL
LIN {X 0,Y 298.661,Z 413.281,A -85,B 0,C 180,E1 -16374.599,E2 -16374.599} C_VEL
LIN {X 0,Y 298.923,Z 413.249,A -85,B 0,C 180,E1 -16378.653,E2 -16378.653} C_VEL
LIN {X 0,Y 298.924,Z 413.248,A -85,B 0,C 180,E1 -16381.347,E2 -16381.347} C_VEL
LIN {X 0,Y 298.799,Z 413.265,A -85,B 0,C 180,E1 -16386.754,E2 -16386.754} C_VEL
LIN {X 0,Y 298.682,Z 413.277,A -85,B 0,C 180,E1 -16389.48,E2 -16389.48} C_VEL
LIN {X 0,Y 298.553,Z 413.291,A -85,B 0,C 180,E1 -16393.615,E2 -16393.615} C_VEL
LIN {X 0,Y 298.55,Z 413.292,A -85,B 0,C 180,E1 -16396.409,E2 -16396.409} C_VEL
LIN {X 0,Y 298.513,Z 413.294,A -85,B 0,C 180,E1 -16399.655,E2 -16399.655} C_VEL
LIN {X 0,Y 298.459,Z 413.304,A -85,B 0,C 180,E1 -16403.598,E2 -16403.598} C_VEL
LIN {X 0,Y 298.493,Z 413.304,A -85,B 0,C 180,E1 -16406.574,E2 -16406.574} C_VEL
LIN {X 0,Y 298.422,Z 413.309,A -85,B 0,C 180,E1 -16409.641,E2 -16409.641} C_VEL
LIN {X 0,Y 298.396,Z 413.314,A -85,B 0,C 180,E1 -16412.8,E2 -16412.8} C_VEL
LIN {X 0,Y 298.447,Z 413.307,A -85,B 0,C 180,E1 -16416.807,E2 -16416.807} C_VEL
LIN {X 0,Y 298.388,Z 413.315,A -85,B 0,C 180,E1 -16421.088,E2 -16421.088} C_VEL
LIN {X 0,Y 298.4,Z 413.314,A -85,B 0,C 180,E1 -16423.103,E2 -16423.103} C_VEL
LIN {X 0,Y 298.404,Z 413.313,A -85,B 0,C 180,E1 -16426.921,E2 -16426.921} C_VEL
LIN {X 0,Y 298.416,Z 413.309,A -85,B 0,C 180,E1 -16431.003,E2 -16431.003} C_VEL
LIN {X 0,Y 298.434,Z 413.307,A -85,B 0,C 180,E1 -16433.932,E2 -16433.932} C_VEL
LIN {X 0,Y 298.395,Z 413.314,A -85,B 0,C 180,E1 -16437.984,E2 -16437.984} C_VEL
LIN {X 0,Y 298.458,Z 413.304,A -85,B 0,C 180,E1 -16441.903,E2 -16441.903} C_VEL
LIN {X 0,Y 298.485,Z 413.303,A -85,B 0,C 180,E1 -16444.924,E2 -16444.924} C_VEL
LIN {X 0,Y 298.46,Z 413.305,A -85,B 0,C 180,E1 -16449.316,E2 -16449.316} C_VEL
LIN {X 0,Y 298.54,Z 413.297,A -85,B 0,C 180,E1 -16452.179,E2 -16452.179} C_VEL
LIN {X 0,Y 298.595,Z 413.289,A -85,B 0,C 180,E1 -16454.994,E2 -16454.994} C_VEL
LIN {X 0,Y 298.595,Z 413.287,A -85,B 0,C 180,E1 -16459.146,E2 -16459.146} C_VEL
LIN {X 0,Y 298.762,Z 413.269,A -85,B 0,C 180,E1 -16461.886,E2 -16461.886} C_VEL
LIN {X 0,Y 298.661,Z 413.281,A -85,B 0,C 180,E1 -16464.598,E2 -16464.598} C_VEL
LIN {X 0,Y 298.924,Z 413.25,A -85,B 0,C 180,E1 -16468.652,E2 -16468.652} C_VEL
